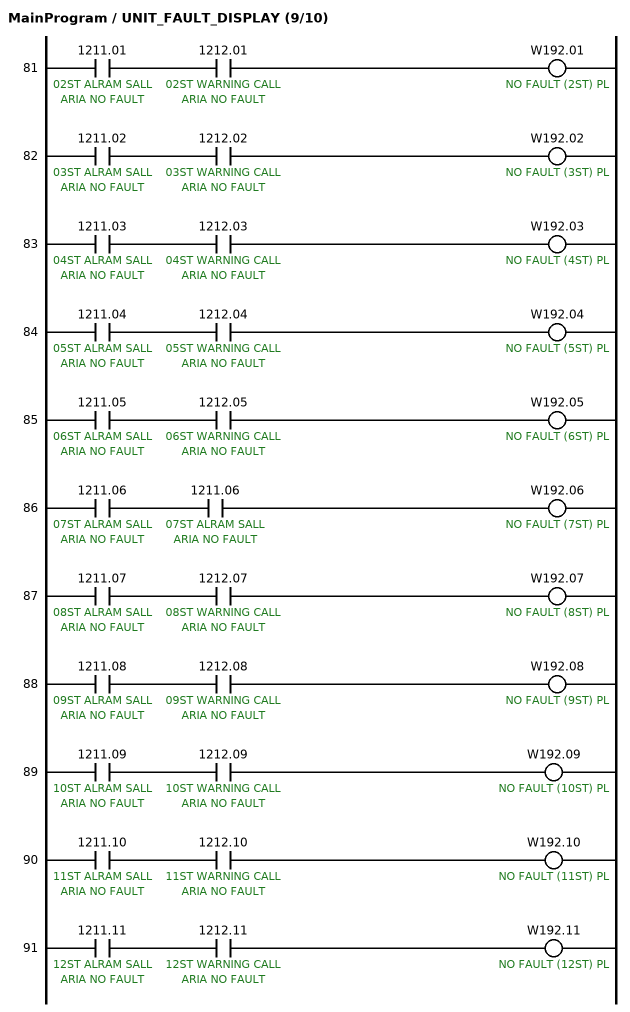
; [picture p120: MainProgram / UNIT_FAULT_DISPLAY, rungs 81-91]
; rung 81
LD 1211.01  ; 02ST ALRAM SALL ARIA NO FAULT
AND 1212.01  ; 02ST WARNING CALL ARIA NO FAULT
OUT W192.01  ; NO FAULT (2ST) PL
; rung 82
LD 1211.02  ; 03ST ALRAM SALL ARIA NO FAULT
AND 1212.02  ; 03ST WARNING CALL ARIA NO FAULT
OUT W192.02  ; NO FAULT (3ST) PL
; rung 83
LD 1211.03  ; 04ST ALRAM SALL ARIA NO FAULT
AND 1212.03  ; 04ST WARNING CALL ARIA NO FAULT
OUT W192.03  ; NO FAULT (4ST) PL
; rung 84
LD 1211.04  ; 05ST ALRAM SALL ARIA NO FAULT
AND 1212.04  ; 05ST WARNING CALL ARIA NO FAULT
OUT W192.04  ; NO FAULT (5ST) PL
; rung 85
LD 1211.05  ; 06ST ALRAM SALL ARIA NO FAULT
AND 1212.05  ; 06ST WARNING CALL ARIA NO FAULT
OUT W192.05  ; NO FAULT (6ST) PL
; rung 86
LD 1211.06  ; 07ST ALRAM SALL ARIA NO FAULT
AND 1211.06  ; 07ST ALRAM SALL ARIA NO FAULT
OUT W192.06  ; NO FAULT (7ST) PL
; rung 87
LD 1211.07  ; 08ST ALRAM SALL ARIA NO FAULT
AND 1212.07  ; 08ST WARNING CALL ARIA NO FAULT
OUT W192.07  ; NO FAULT (8ST) PL
; rung 88
LD 1211.08  ; 09ST ALRAM SALL ARIA NO FAULT
AND 1212.08  ; 09ST WARNING CALL ARIA NO FAULT
OUT W192.08  ; NO FAULT (9ST) PL
; rung 89
LD 1211.09  ; 10ST ALRAM SALL ARIA NO FAULT
AND 1212.09  ; 10ST WARNING CALL ARIA NO FAULT
OUT W192.09  ; NO FAULT (10ST) PL
; rung 90
LD 1211.10  ; 11ST ALRAM SALL ARIA NO FAULT
AND 1212.10  ; 11ST WARNING CALL ARIA NO FAULT
OUT W192.10  ; NO FAULT (11ST) PL
; rung 91
LD 1211.11  ; 12ST ALRAM SALL ARIA NO FAULT
AND 1212.11  ; 12ST WARNING CALL ARIA NO FAULT
OUT W192.11  ; NO FAULT (12ST) PL

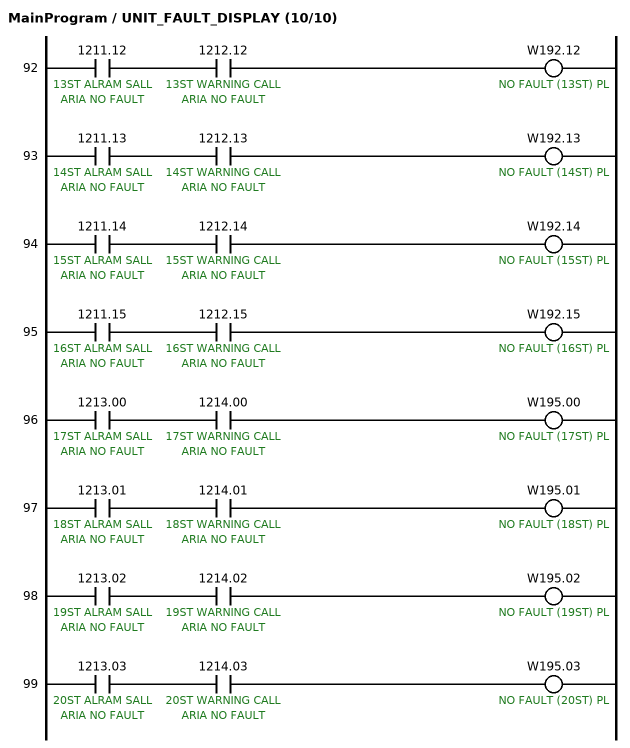
; rung 92
LD 1211.12  ; 13ST ALRAM SALL ARIA NO FAULT
AND 1212.12  ; 13ST WARNING CALL ARIA NO FAULT
OUT W192.12  ; NO FAULT (13ST) PL
; rung 93
LD 1211.13  ; 14ST ALRAM SALL ARIA NO FAULT
AND 1212.13  ; 14ST WARNING CALL ARIA NO FAULT
OUT W192.13  ; NO FAULT (14ST) PL
; rung 94
LD 1211.14  ; 15ST ALRAM SALL ARIA NO FAULT
AND 1212.14  ; 15ST WARNING CALL ARIA NO FAULT
OUT W192.14  ; NO FAULT (15ST) PL
; rung 95
LD 1211.15  ; 16ST ALRAM SALL ARIA NO FAULT
AND 1212.15  ; 16ST WARNING CALL ARIA NO FAULT
OUT W192.15  ; NO FAULT (16ST) PL
; rung 96
LD 1213.00  ; 17ST ALRAM SALL ARIA NO FAULT
AND 1214.00  ; 17ST WARNING CALL ARIA NO FAULT
OUT W195.00  ; NO FAULT (17ST) PL
; rung 97
LD 1213.01  ; 18ST ALRAM SALL ARIA NO FAULT
AND 1214.01  ; 18ST WARNING CALL ARIA NO FAULT
OUT W195.01  ; NO FAULT (18ST) PL
; rung 98
LD 1213.02  ; 19ST ALRAM SALL ARIA NO FAULT
AND 1214.02  ; 19ST WARNING CALL ARIA NO FAULT
OUT W195.02  ; NO FAULT (19ST) PL
; rung 99
LD 1213.03  ; 20ST ALRAM SALL ARIA NO FAULT
AND 1214.03  ; 20ST WARNING CALL ARIA NO FAULT
OUT W195.03  ; NO FAULT (20ST) PL

### Section FAULT_DISPLAY

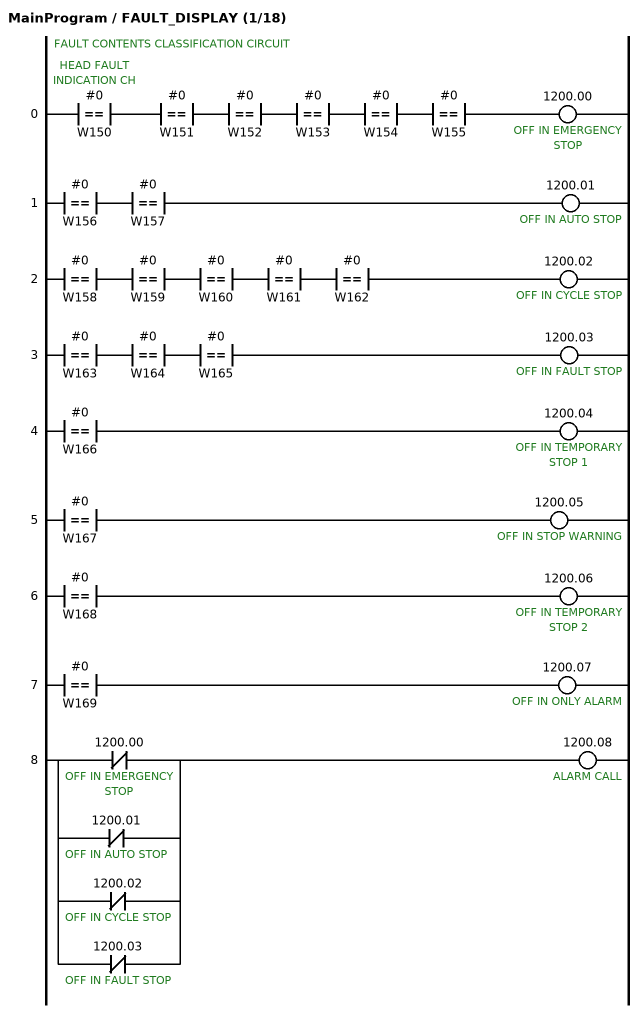
; rung 0: FAULT CONTENTS CLASSIFICATION CIRCUIT
LD=(300) #0 W150  ; HEAD FAULT INDICATION CH
AND=(300) #0 W151
AND=(300) #0 W152
AND=(300) #0 W153
AND=(300) #0 W154
AND=(300) #0 W155
OUT 1200.00  ; OFF IN EMERGENCY STOP
; rung 1
LD=(300) #0 W156
AND=(300) #0 W157
OUT 1200.01  ; OFF IN AUTO STOP
; rung 2
LD=(300) #0 W158
AND=(300) #0 W159
AND=(300) #0 W160
AND=(300) #0 W161
AND=(300) #0 W162
OUT 1200.02  ; OFF IN CYCLE STOP
; rung 3
LD=(300) #0 W163
AND=(300) #0 W164
AND=(300) #0 W165
OUT 1200.03  ; OFF IN FAULT STOP
; rung 4
LD=(300) #0 W166
OUT 1200.04  ; OFF IN TEMPORARY STOP 1
; rung 5
LD=(300) #0 W167
OUT 1200.05  ; OFF IN STOP WARNING
; rung 6
LD=(300) #0 W168
OUT 1200.06  ; OFF IN TEMPORARY STOP 2
; rung 7
LD=(300) #0 W169
OUT 1200.07  ; OFF IN ONLY ALARM
; rung 8
LDNOT 1200.00  ; OFF IN EMERGENCY STOP
ORNOT 1200.01  ; OFF IN AUTO STOP
ORNOT 1200.02  ; OFF IN CYCLE STOP
ORNOT 1200.03  ; OFF IN FAULT STOP
OUT 1200.08  ; ALARM CALL

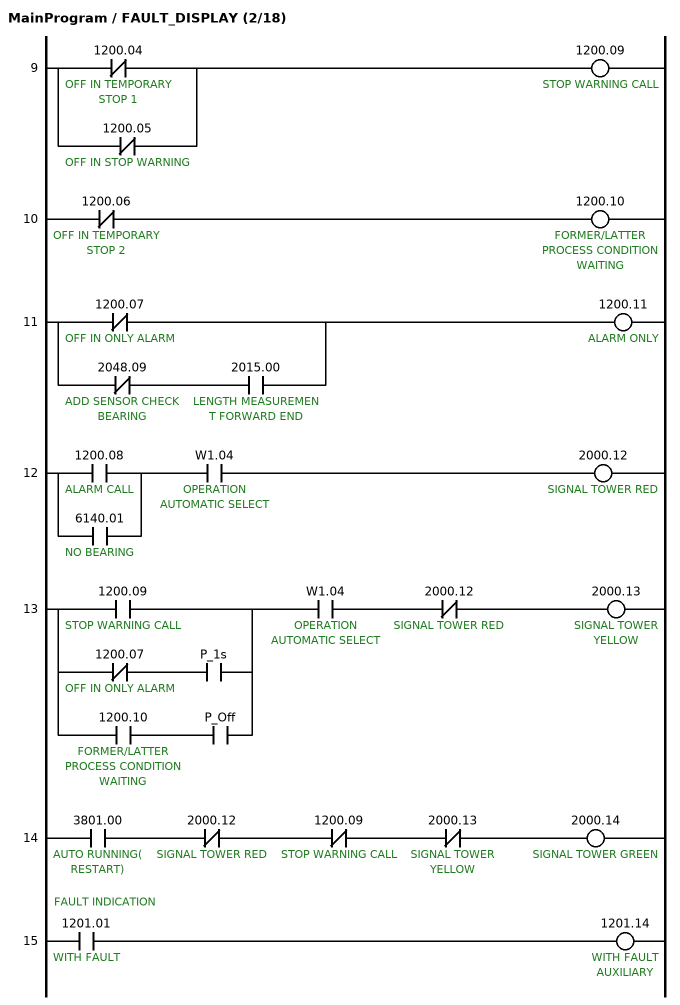
; rung 9
LDNOT 1200.04  ; OFF IN TEMPORARY STOP 1
ORNOT 1200.05  ; OFF IN STOP WARNING
OUT 1200.09  ; STOP WARNING CALL
; rung 10
LDNOT 1200.06  ; OFF IN TEMPORARY STOP 2
OUT 1200.10  ; FORMER/LATTER PROCESS CONDITION WAITING
; rung 11
LDNOT 1200.07  ; OFF IN ONLY ALARM
LDNOT 2048.09  ; ADD SENSOR CHECK BEARING
AND 2015.00  ; LENGTH MEASUREMENT FORWARD END
ORLD
OUT 1200.11  ; ALARM ONLY
; rung 12
LD 1200.08  ; ALARM CALL
OR 6140.01  ; NO BEARING
AND W1.04  ; OPERATION AUTOMATIC SELECT
OUT 2000.12  ; SIGNAL TOWER RED
; rung 13
LD 1200.09  ; STOP WARNING CALL
LDNOT 1200.07  ; OFF IN ONLY ALARM
AND P_1s
ORLD
LD 1200.10  ; FORMER/LATTER PROCESS CONDITION WAITING
AND P_Off
ORLD
AND W1.04  ; OPERATION AUTOMATIC SELECT
ANDNOT 2000.12  ; SIGNAL TOWER RED
OUT 2000.13  ; SIGNAL TOWER YELLOW
; rung 14
LD 3801.00  ; AUTO RUNNING(RESTART)
ANDNOT 2000.12  ; SIGNAL TOWER RED
ANDNOT 1200.09  ; STOP WARNING CALL
ANDNOT 2000.13  ; SIGNAL TOWER YELLOW
OUT 2000.14  ; SIGNAL TOWER GREEN
; rung 15: FAULT INDICATION
LD 1201.01  ; WITH FAULT
OUT 1201.14  ; WITH FAULT AUXILIARY

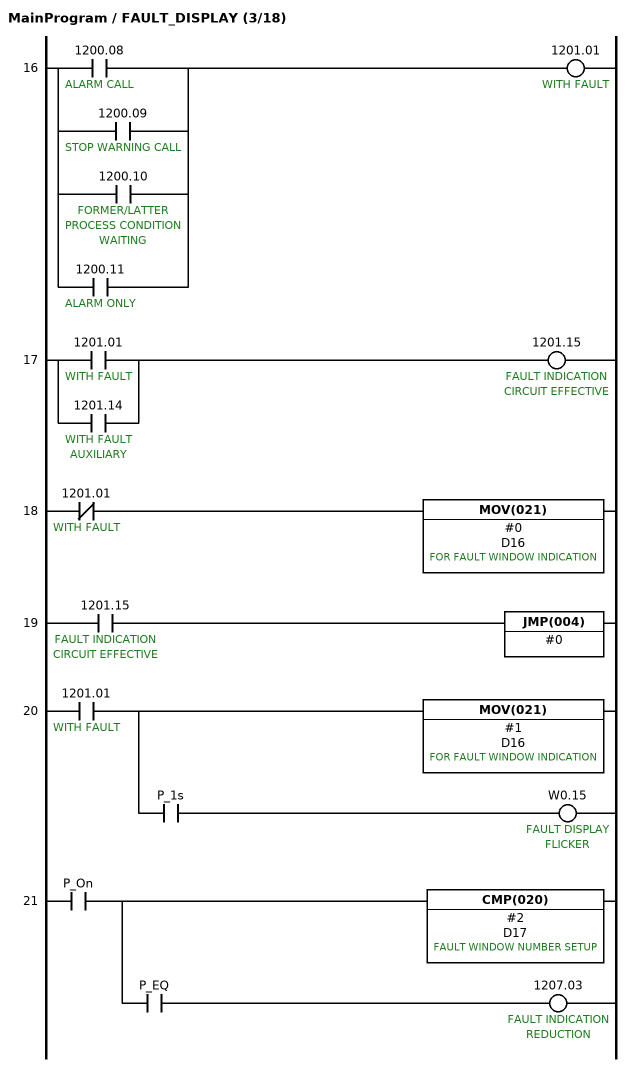
; rung 16
LD 1200.08  ; ALARM CALL
OR 1200.09  ; STOP WARNING CALL
OR 1200.10  ; FORMER/LATTER PROCESS CONDITION WAITING
OR 1200.11  ; ALARM ONLY
OUT 1201.01  ; WITH FAULT
; rung 17
LD 1201.01  ; WITH FAULT
OR 1201.14  ; WITH FAULT AUXILIARY
OUT 1201.15  ; FAULT INDICATION CIRCUIT EFFECTIVE
; rung 18
LDNOT 1201.01  ; WITH FAULT
MOV(021) #0 D16  ; FOR FAULT WINDOW INDICATION  // WITH NO FAULT WINDOW DISPLAY
; rung 19
LD 1201.15  ; FAULT INDICATION CIRCUIT EFFECTIVE
JMP(004) #0
; rung 20
LD 1201.01  ; WITH FAULT
MOV(021) #1 D16  ; FOR FAULT WINDOW INDICATION  // FAULT WINDOW DISPLAY
AND P_1s
OUT W0.15  ; FAULT DISPLAY FLICKER
; rung 21
LD P_On
CMP(020) #2 D17  ; FAULT WINDOW NUMBER SETUP
AND P_EQ
OUT 1207.03  ; FAULT INDICATION REDUCTION

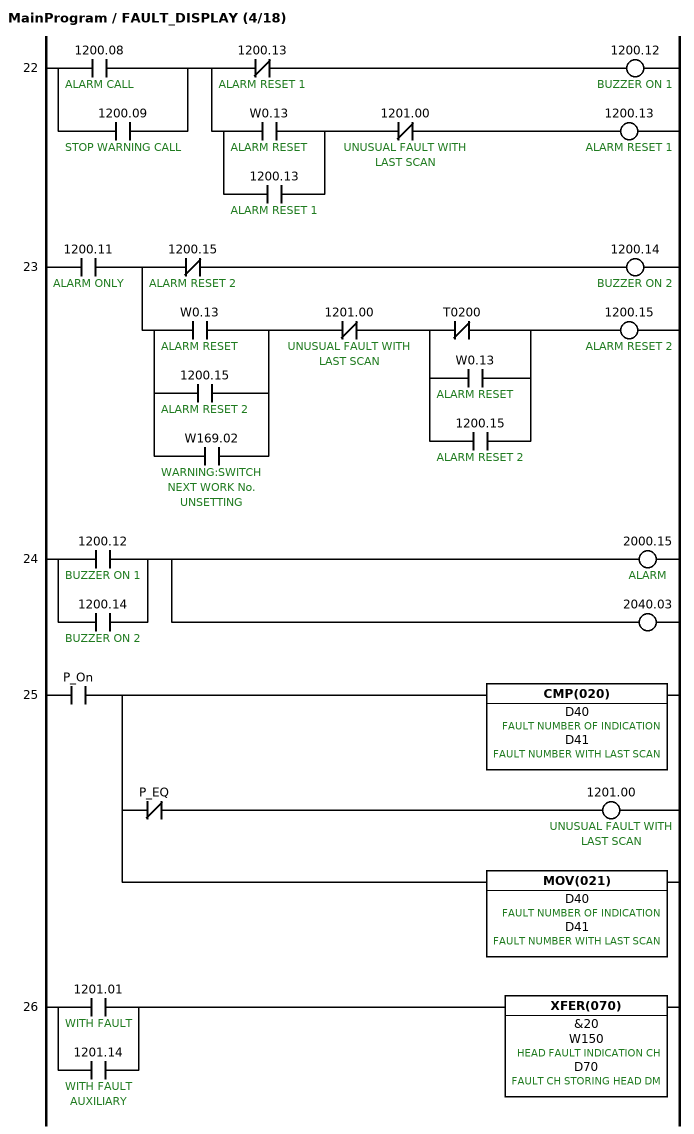
; rung 22
LD 1200.08  ; ALARM CALL
OR 1200.09  ; STOP WARNING CALL
OUT TR0
ANDNOT 1200.13  ; ALARM RESET 1
OUT 1200.12  ; BUZZER ON 1
LD TR0
LD W0.13  ; ALARM RESET
OR 1200.13  ; ALARM RESET 1
ANDLD
ANDNOT 1201.00  ; UNUSUAL FAULT WITH LAST SCAN
OUT 1200.13  ; ALARM RESET 1
; rung 23
LD 1200.11  ; ALARM ONLY
OUT TR0
ANDNOT 1200.15  ; ALARM RESET 2
OUT 1200.14  ; BUZZER ON 2
LD TR0
LD W0.13  ; ALARM RESET
OR 1200.15  ; ALARM RESET 2
OR W169.02  ; WARNING:SWITCH NEXT WORK No. UNSETTING
ANDLD
ANDNOT 1201.00  ; UNUSUAL FAULT WITH LAST SCAN
LDNOT T0200
OR W0.13  ; ALARM RESET
OR 1200.15  ; ALARM RESET 2
ANDLD
OUT 1200.15  ; ALARM RESET 2
; rung 24
LD 1200.12  ; BUZZER ON 1
OR 1200.14  ; BUZZER ON 2
OUT 2000.15  ; ALARM
OUT 2040.03
; rung 25
LD P_On
OUT TR0
CMP(020) D40 D41  ; FAULT NUMBER OF INDICATION, FAULT NUMBER WITH LAST SCAN  // FAULT NUMBER COMPARISON
ANDNOT P_EQ
OUT 1201.00  ; UNUSUAL FAULT WITH LAST SCAN
LD TR0
MOV(021) D40 D41  ; FAULT NUMBER OF INDICATION, FAULT NUMBER WITH LAST SCAN  // FAULT NUMBER TRANSMISSION FOR NEXT SCAN COMPARISON
; rung 26
LD 1201.01  ; WITH FAULT
OR 1201.14  ; WITH FAULT AUXILIARY
XFER(070) &20 W150 D70  ; HEAD FAULT INDICATION CH, FAULT CH STORING HEAD DM  // ALL FAULT CH ARE TRANSMISSION TO DM0070-89

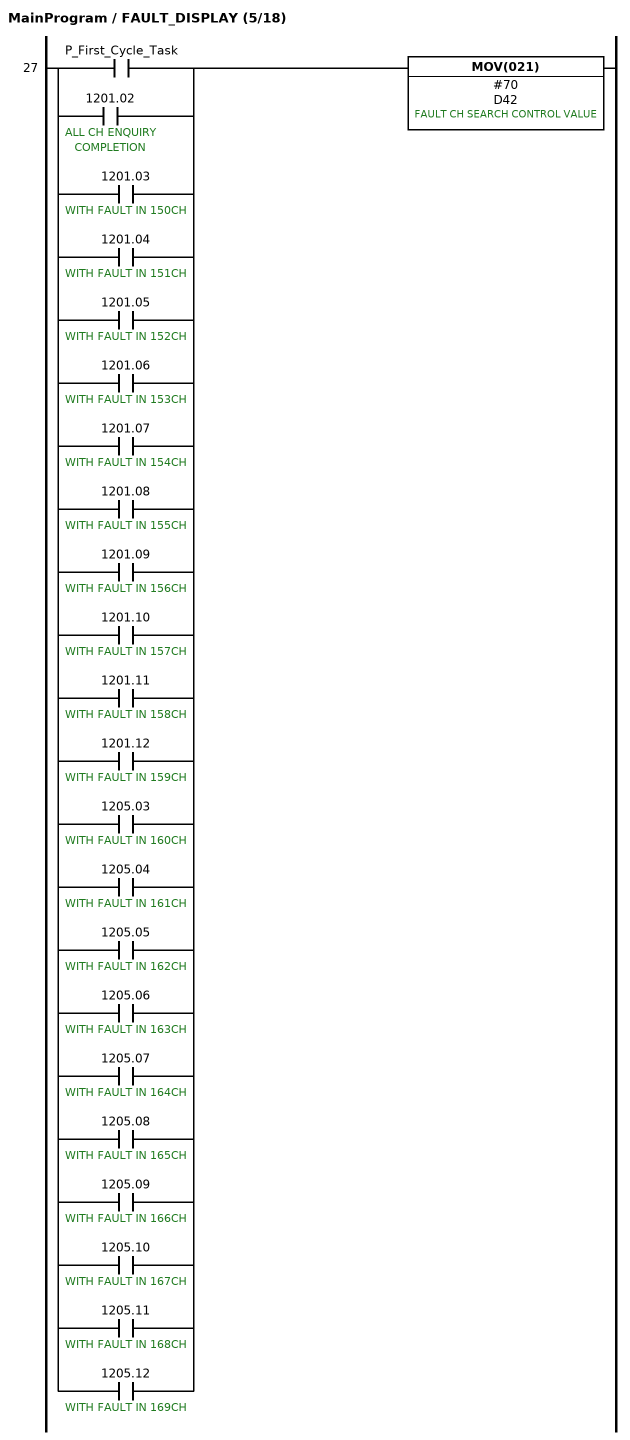
; rung 27
LD P_First_Cycle_Task
OR 1201.02  ; ALL CH ENQUIRY COMPLETION
OR 1201.03  ; WITH FAULT IN 150CH
OR 1201.04  ; WITH FAULT IN 151CH
OR 1201.05  ; WITH FAULT IN 152CH
OR 1201.06  ; WITH FAULT IN 153CH
OR 1201.07  ; WITH FAULT IN 154CH
OR 1201.08  ; WITH FAULT IN 155CH
OR 1201.09  ; WITH FAULT IN 156CH
OR 1201.10  ; WITH FAULT IN 157CH
OR 1201.11  ; WITH FAULT IN 158CH
OR 1201.12  ; WITH FAULT IN 159CH
OR 1205.03  ; WITH FAULT IN 160CH
OR 1205.04  ; WITH FAULT IN 161CH
OR 1205.05  ; WITH FAULT IN 162CH
OR 1205.06  ; WITH FAULT IN 163CH
OR 1205.07  ; WITH FAULT IN 164CH
OR 1205.08  ; WITH FAULT IN 165CH
OR 1205.09  ; WITH FAULT IN 166CH
OR 1205.10  ; WITH FAULT IN 167CH
OR 1205.11  ; WITH FAULT IN 168CH
OR 1205.12  ; WITH FAULT IN 169CH
MOV(021) #70 D42  ; FAULT CH SEARCH CONTROL VALUE  // FOR FAULT CH REFERENCE,CONTORL VALUE INITIALIZATION

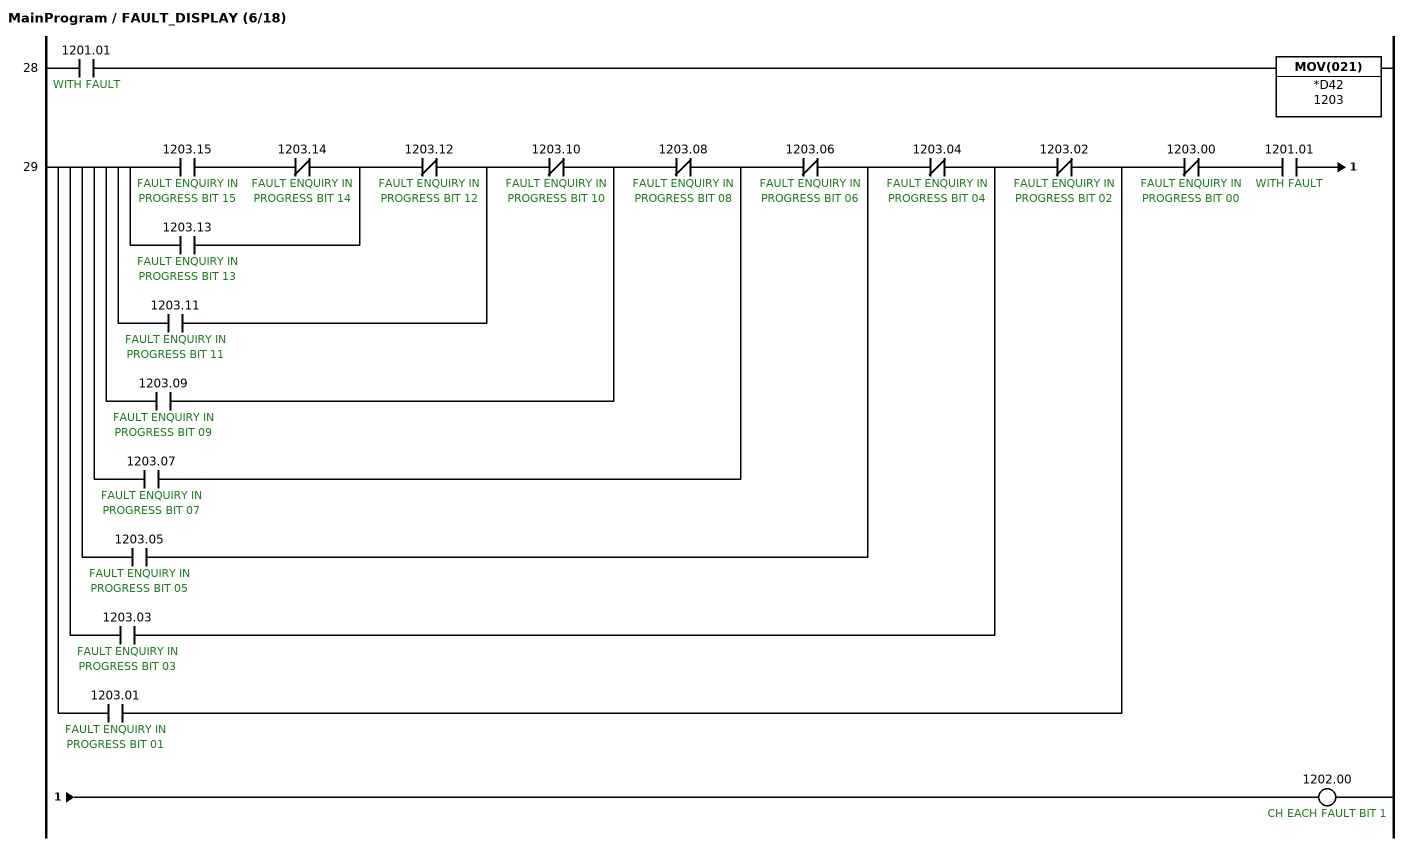
; rung 28
LD 1201.01  ; WITH FAULT
MOV(021) *D42 1203  // FAULT BIT IN CH IS TRANSMISSION DURING REFERENCE
; rung 29
LD 1203.15  ; FAULT ENQUIRY IN PROGRESS BIT 15
ANDNOT 1203.14  ; FAULT ENQUIRY IN PROGRESS BIT 14
OR 1203.13  ; FAULT ENQUIRY IN PROGRESS BIT 13
ANDNOT 1203.12  ; FAULT ENQUIRY IN PROGRESS BIT 12
OR 1203.11  ; FAULT ENQUIRY IN PROGRESS BIT 11
ANDNOT 1203.10  ; FAULT ENQUIRY IN PROGRESS BIT 10
OR 1203.09  ; FAULT ENQUIRY IN PROGRESS BIT 09
ANDNOT 1203.08  ; FAULT ENQUIRY IN PROGRESS BIT 08
OR 1203.07  ; FAULT ENQUIRY IN PROGRESS BIT 07
ANDNOT 1203.06  ; FAULT ENQUIRY IN PROGRESS BIT 06
OR 1203.05  ; FAULT ENQUIRY IN PROGRESS BIT 05
ANDNOT 1203.04  ; FAULT ENQUIRY IN PROGRESS BIT 04
OR 1203.03  ; FAULT ENQUIRY IN PROGRESS BIT 03
ANDNOT 1203.02  ; FAULT ENQUIRY IN PROGRESS BIT 02
OR 1203.01  ; FAULT ENQUIRY IN PROGRESS BIT 01
ANDNOT 1203.00  ; FAULT ENQUIRY IN PROGRESS BIT 00
AND 1201.01  ; WITH FAULT
OUT 1202.00  ; CH EACH FAULT BIT 1

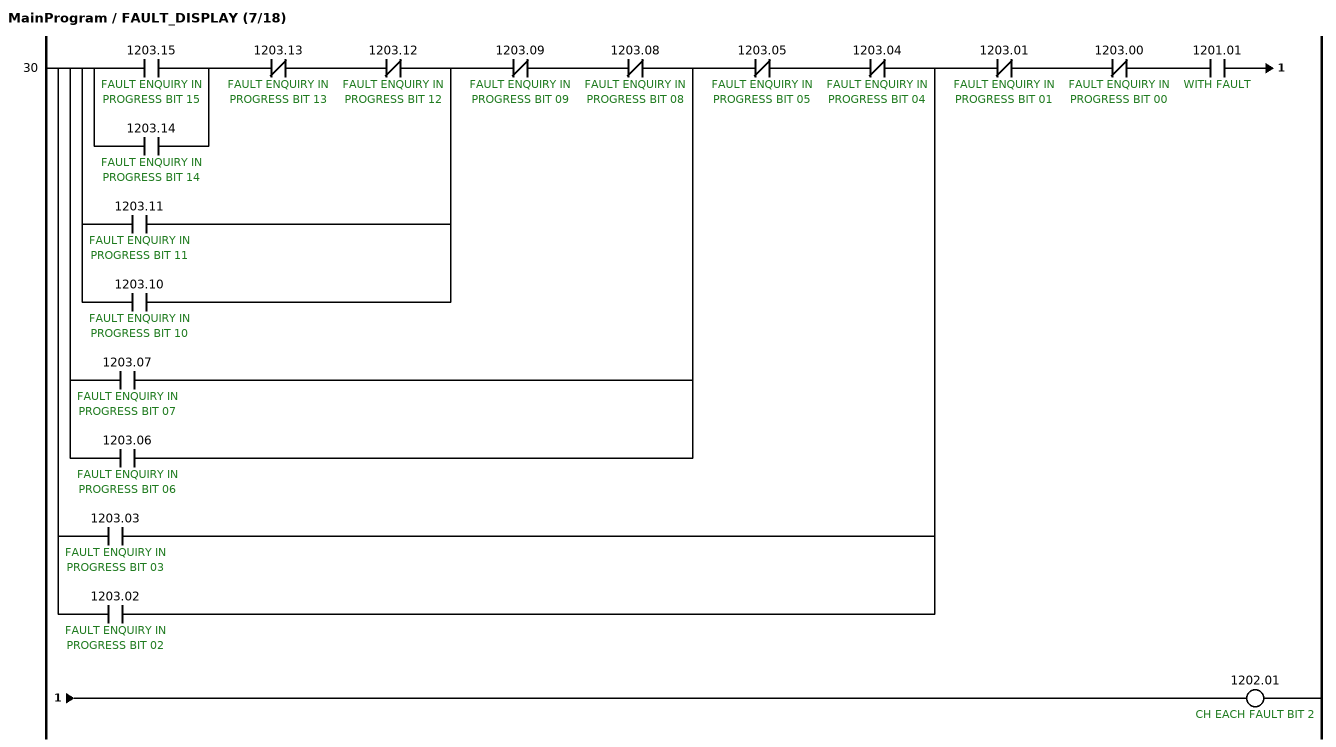
; rung 30
LD 1203.15  ; FAULT ENQUIRY IN PROGRESS BIT 15
OR 1203.14  ; FAULT ENQUIRY IN PROGRESS BIT 14
ANDNOT 1203.13  ; FAULT ENQUIRY IN PROGRESS BIT 13
ANDNOT 1203.12  ; FAULT ENQUIRY IN PROGRESS BIT 12
OR 1203.11  ; FAULT ENQUIRY IN PROGRESS BIT 11
OR 1203.10  ; FAULT ENQUIRY IN PROGRESS BIT 10
ANDNOT 1203.09  ; FAULT ENQUIRY IN PROGRESS BIT 09
ANDNOT 1203.08  ; FAULT ENQUIRY IN PROGRESS BIT 08
OR 1203.07  ; FAULT ENQUIRY IN PROGRESS BIT 07
OR 1203.06  ; FAULT ENQUIRY IN PROGRESS BIT 06
ANDNOT 1203.05  ; FAULT ENQUIRY IN PROGRESS BIT 05
ANDNOT 1203.04  ; FAULT ENQUIRY IN PROGRESS BIT 04
OR 1203.03  ; FAULT ENQUIRY IN PROGRESS BIT 03
OR 1203.02  ; FAULT ENQUIRY IN PROGRESS BIT 02
ANDNOT 1203.01  ; FAULT ENQUIRY IN PROGRESS BIT 01
ANDNOT 1203.00  ; FAULT ENQUIRY IN PROGRESS BIT 00
AND 1201.01  ; WITH FAULT
OUT 1202.01  ; CH EACH FAULT BIT 2

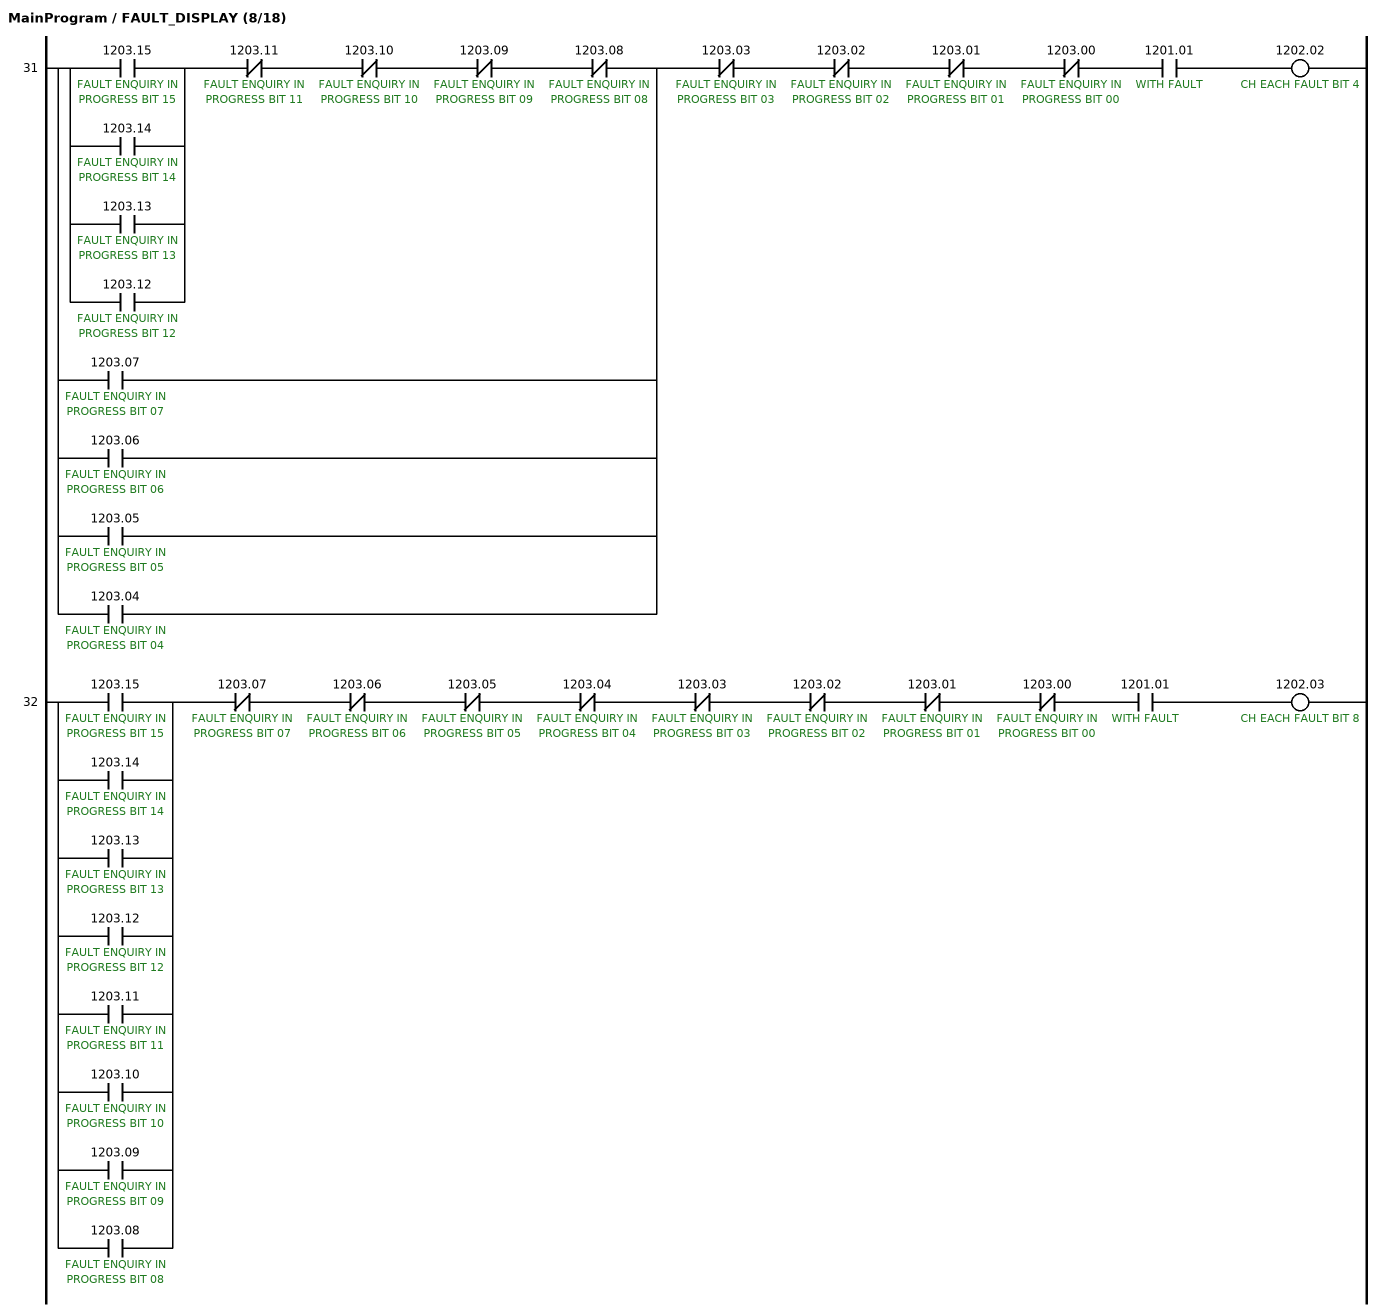
; rung 31
LD 1203.15  ; FAULT ENQUIRY IN PROGRESS BIT 15
OR 1203.14  ; FAULT ENQUIRY IN PROGRESS BIT 14
OR 1203.13  ; FAULT ENQUIRY IN PROGRESS BIT 13
OR 1203.12  ; FAULT ENQUIRY IN PROGRESS BIT 12
ANDNOT 1203.11  ; FAULT ENQUIRY IN PROGRESS BIT 11
ANDNOT 1203.10  ; FAULT ENQUIRY IN PROGRESS BIT 10
ANDNOT 1203.09  ; FAULT ENQUIRY IN PROGRESS BIT 09
ANDNOT 1203.08  ; FAULT ENQUIRY IN PROGRESS BIT 08
OR 1203.07  ; FAULT ENQUIRY IN PROGRESS BIT 07
OR 1203.06  ; FAULT ENQUIRY IN PROGRESS BIT 06
OR 1203.05  ; FAULT ENQUIRY IN PROGRESS BIT 05
OR 1203.04  ; FAULT ENQUIRY IN PROGRESS BIT 04
ANDNOT 1203.03  ; FAULT ENQUIRY IN PROGRESS BIT 03
ANDNOT 1203.02  ; FAULT ENQUIRY IN PROGRESS BIT 02
ANDNOT 1203.01  ; FAULT ENQUIRY IN PROGRESS BIT 01
ANDNOT 1203.00  ; FAULT ENQUIRY IN PROGRESS BIT 00
AND 1201.01  ; WITH FAULT
OUT 1202.02  ; CH EACH FAULT BIT 4
; rung 32
LD 1203.15  ; FAULT ENQUIRY IN PROGRESS BIT 15
OR 1203.14  ; FAULT ENQUIRY IN PROGRESS BIT 14
OR 1203.13  ; FAULT ENQUIRY IN PROGRESS BIT 13
OR 1203.12  ; FAULT ENQUIRY IN PROGRESS BIT 12
OR 1203.11  ; FAULT ENQUIRY IN PROGRESS BIT 11
OR 1203.10  ; FAULT ENQUIRY IN PROGRESS BIT 10
OR 1203.09  ; FAULT ENQUIRY IN PROGRESS BIT 09
OR 1203.08  ; FAULT ENQUIRY IN PROGRESS BIT 08
ANDNOT 1203.07  ; FAULT ENQUIRY IN PROGRESS BIT 07
ANDNOT 1203.06  ; FAULT ENQUIRY IN PROGRESS BIT 06
ANDNOT 1203.05  ; FAULT ENQUIRY IN PROGRESS BIT 05
ANDNOT 1203.04  ; FAULT ENQUIRY IN PROGRESS BIT 04
ANDNOT 1203.03  ; FAULT ENQUIRY IN PROGRESS BIT 03
ANDNOT 1203.02  ; FAULT ENQUIRY IN PROGRESS BIT 02
ANDNOT 1203.01  ; FAULT ENQUIRY IN PROGRESS BIT 01
ANDNOT 1203.00  ; FAULT ENQUIRY IN PROGRESS BIT 00
AND 1201.01  ; WITH FAULT
OUT 1202.03  ; CH EACH FAULT BIT 8

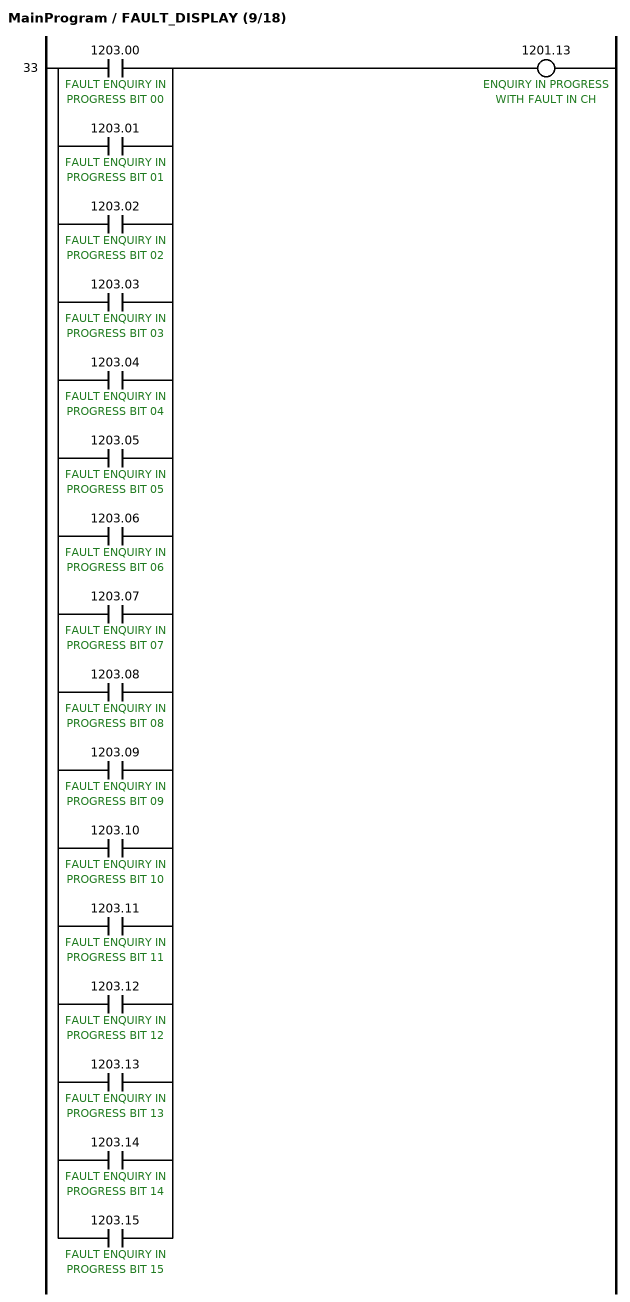
; rung 33
LD 1203.00  ; FAULT ENQUIRY IN PROGRESS BIT 00
OR 1203.01  ; FAULT ENQUIRY IN PROGRESS BIT 01
OR 1203.02  ; FAULT ENQUIRY IN PROGRESS BIT 02
OR 1203.03  ; FAULT ENQUIRY IN PROGRESS BIT 03
OR 1203.04  ; FAULT ENQUIRY IN PROGRESS BIT 04
OR 1203.05  ; FAULT ENQUIRY IN PROGRESS BIT 05
OR 1203.06  ; FAULT ENQUIRY IN PROGRESS BIT 06
OR 1203.07  ; FAULT ENQUIRY IN PROGRESS BIT 07
OR 1203.08  ; FAULT ENQUIRY IN PROGRESS BIT 08
OR 1203.09  ; FAULT ENQUIRY IN PROGRESS BIT 09
OR 1203.10  ; FAULT ENQUIRY IN PROGRESS BIT 10
OR 1203.11  ; FAULT ENQUIRY IN PROGRESS BIT 11
OR 1203.12  ; FAULT ENQUIRY IN PROGRESS BIT 12
OR 1203.13  ; FAULT ENQUIRY IN PROGRESS BIT 13
OR 1203.14  ; FAULT ENQUIRY IN PROGRESS BIT 14
OR 1203.15  ; FAULT ENQUIRY IN PROGRESS BIT 15
OUT 1201.13  ; ENQUIRY IN PROGRESS WITH FAULT IN CH

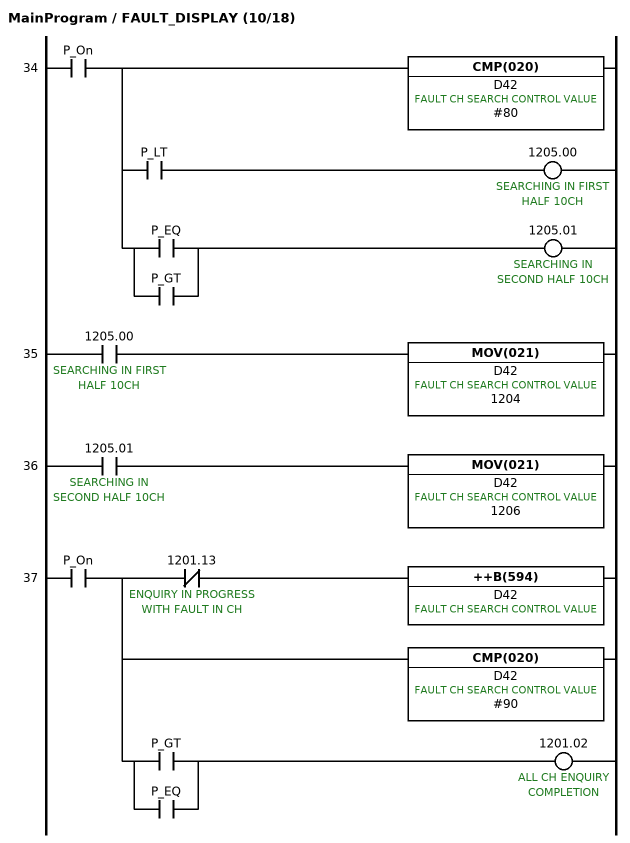
; rung 34
LD P_On
OUT TR0
CMP(020) D42 #80  ; FAULT CH SEARCH CONTROL VALUE
AND P_LT
OUT 1205.00  ; SEARCHING IN FIRST HALF 10CH
LD TR0
LD P_EQ
OR P_GT
ANDLD
OUT 1205.01  ; SEARCHING IN SECOND HALF 10CH
; rung 35
LD 1205.00  ; SEARCHING IN FIRST HALF 10CH
MOV(021) D42 1204  ; FAULT CH SEARCH CONTROL VALUE  // THE CH NUMBER WHEN BEING RETRIEVING IT IS FORWARDED.
; rung 36
LD 1205.01  ; SEARCHING IN SECOND HALF 10CH
MOV(021) D42 1206  ; FAULT CH SEARCH CONTROL VALUE  // THE CH NUMBER WHEN BEING RETRIEVING IT IS FORWARDED.
; rung 37
LD P_On
OUT TR0
ANDNOT 1201.13  ; ENQUIRY IN PROGRESS WITH FAULT IN CH
++B(594) D42  ; FAULT CH SEARCH CONTROL VALUE  // FOR REFERENCE FAULT CH,CONTROL VALUE +1
LD TR0
CMP(020) D42 #90  ; FAULT CH SEARCH CONTROL VALUE  // 90 OR MORE CONTROL VALUES FOR REFERENCE FAULT CH
LD P_GT
OR P_EQ
ANDLD
OUT 1201.02  ; ALL CH ENQUIRY COMPLETION

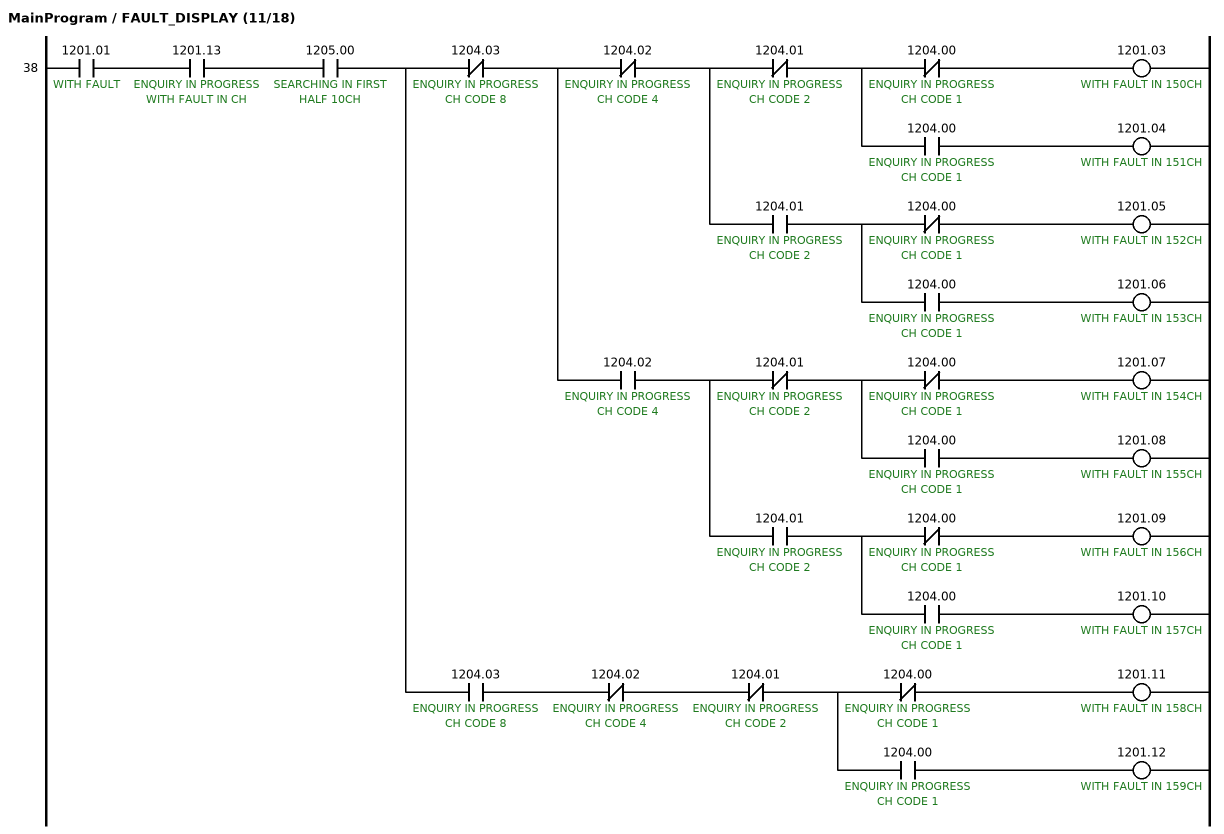
; rung 38
LD 1201.01  ; WITH FAULT
AND 1201.13  ; ENQUIRY IN PROGRESS WITH FAULT IN CH
AND 1205.00  ; SEARCHING IN FIRST HALF 10CH
OUT TR0
ANDNOT 1204.03  ; ENQUIRY IN PROGRESS CH CODE 8
OUT TR1
ANDNOT 1204.02  ; ENQUIRY IN PROGRESS CH CODE 4
OUT TR2
ANDNOT 1204.01  ; ENQUIRY IN PROGRESS CH CODE 2
OUT TR3
ANDNOT 1204.00  ; ENQUIRY IN PROGRESS CH CODE 1
OUT 1201.03  ; WITH FAULT IN 150CH
LD TR3
AND 1204.00  ; ENQUIRY IN PROGRESS CH CODE 1
OUT 1201.04  ; WITH FAULT IN 151CH
LD TR2
AND 1204.01  ; ENQUIRY IN PROGRESS CH CODE 2
OUT TR2
ANDNOT 1204.00  ; ENQUIRY IN PROGRESS CH CODE 1
OUT 1201.05  ; WITH FAULT IN 152CH
LD TR2
AND 1204.00  ; ENQUIRY IN PROGRESS CH CODE 1
OUT 1201.06  ; WITH FAULT IN 153CH
LD TR1
AND 1204.02  ; ENQUIRY IN PROGRESS CH CODE 4
OUT TR1
ANDNOT 1204.01  ; ENQUIRY IN PROGRESS CH CODE 2
OUT TR2
ANDNOT 1204.00  ; ENQUIRY IN PROGRESS CH CODE 1
OUT 1201.07  ; WITH FAULT IN 154CH
LD TR2
AND 1204.00  ; ENQUIRY IN PROGRESS CH CODE 1
OUT 1201.08  ; WITH FAULT IN 155CH
LD TR1
AND 1204.01  ; ENQUIRY IN PROGRESS CH CODE 2
OUT TR1
ANDNOT 1204.00  ; ENQUIRY IN PROGRESS CH CODE 1
OUT 1201.09  ; WITH FAULT IN 156CH
LD TR1
AND 1204.00  ; ENQUIRY IN PROGRESS CH CODE 1
OUT 1201.10  ; WITH FAULT IN 157CH
LD TR0
AND 1204.03  ; ENQUIRY IN PROGRESS CH CODE 8
ANDNOT 1204.02  ; ENQUIRY IN PROGRESS CH CODE 4
ANDNOT 1204.01  ; ENQUIRY IN PROGRESS CH CODE 2
OUT TR0
ANDNOT 1204.00  ; ENQUIRY IN PROGRESS CH CODE 1
OUT 1201.11  ; WITH FAULT IN 158CH
LD TR0
AND 1204.00  ; ENQUIRY IN PROGRESS CH CODE 1
OUT 1201.12  ; WITH FAULT IN 159CH

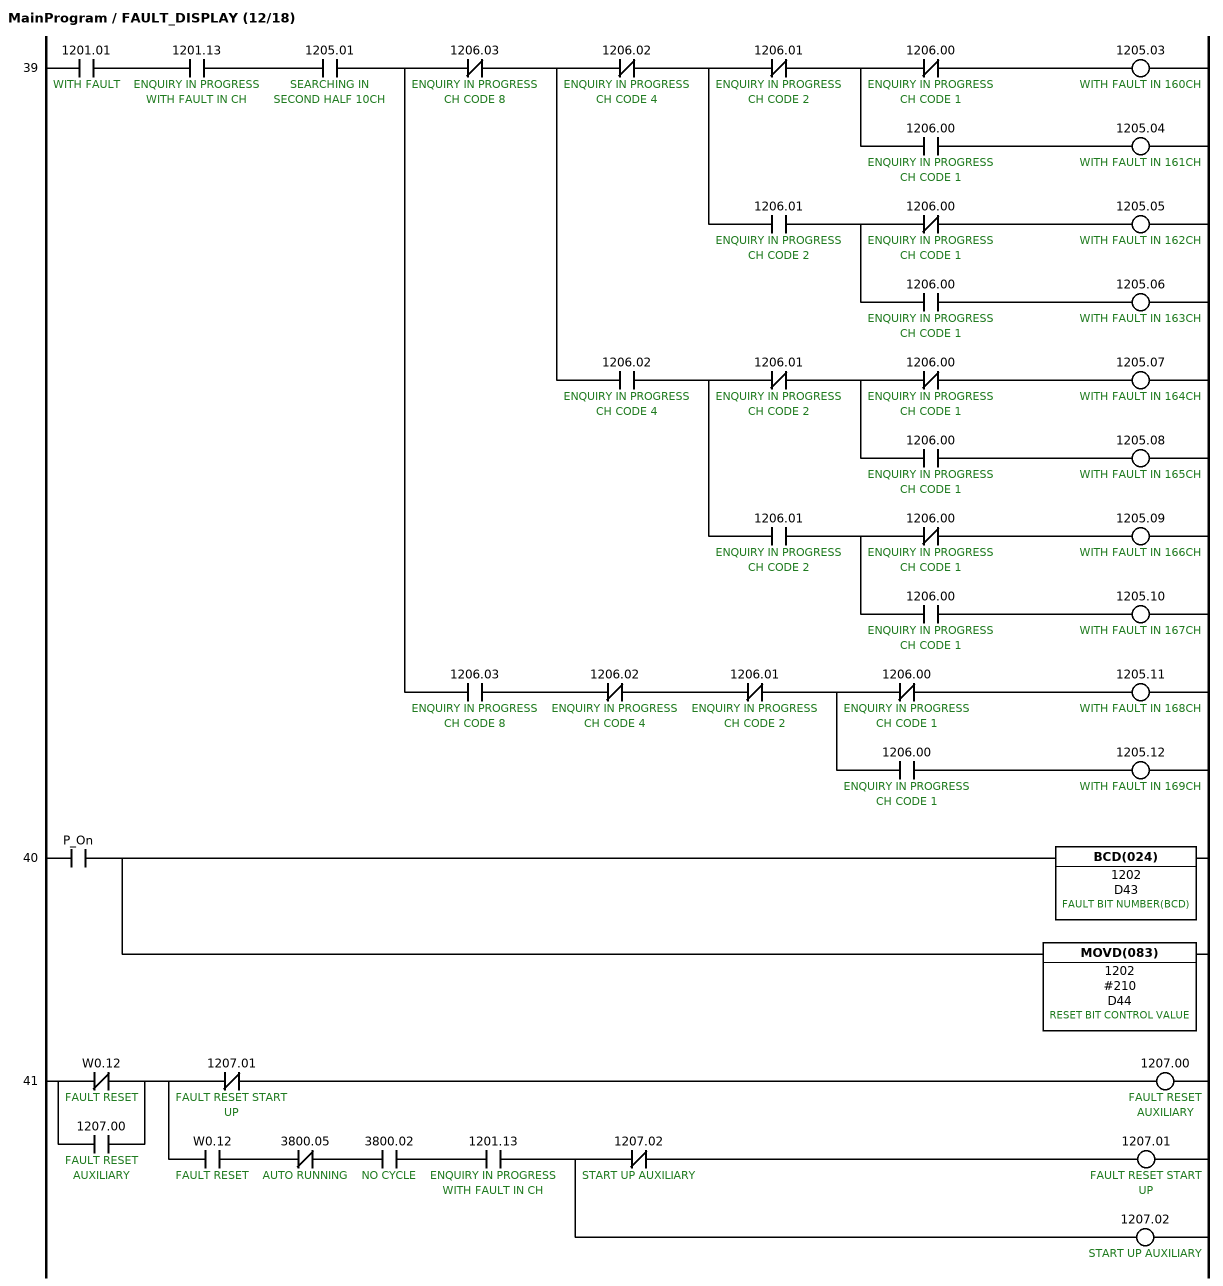
; rung 39
LD 1201.01  ; WITH FAULT
AND 1201.13  ; ENQUIRY IN PROGRESS WITH FAULT IN CH
AND 1205.01  ; SEARCHING IN SECOND HALF 10CH
OUT TR0
ANDNOT 1206.03  ; ENQUIRY IN PROGRESS CH CODE 8
OUT TR1
ANDNOT 1206.02  ; ENQUIRY IN PROGRESS CH CODE 4
OUT TR2
ANDNOT 1206.01  ; ENQUIRY IN PROGRESS CH CODE 2
OUT TR3
ANDNOT 1206.00  ; ENQUIRY IN PROGRESS CH CODE 1
OUT 1205.03  ; WITH FAULT IN 160CH
LD TR3
AND 1206.00  ; ENQUIRY IN PROGRESS CH CODE 1
OUT 1205.04  ; WITH FAULT IN 161CH
LD TR2
AND 1206.01  ; ENQUIRY IN PROGRESS CH CODE 2
OUT TR2
ANDNOT 1206.00  ; ENQUIRY IN PROGRESS CH CODE 1
OUT 1205.05  ; WITH FAULT IN 162CH
LD TR2
AND 1206.00  ; ENQUIRY IN PROGRESS CH CODE 1
OUT 1205.06  ; WITH FAULT IN 163CH
LD TR1
AND 1206.02  ; ENQUIRY IN PROGRESS CH CODE 4
OUT TR1
ANDNOT 1206.01  ; ENQUIRY IN PROGRESS CH CODE 2
OUT TR2
ANDNOT 1206.00  ; ENQUIRY IN PROGRESS CH CODE 1
OUT 1205.07  ; WITH FAULT IN 164CH
LD TR2
AND 1206.00  ; ENQUIRY IN PROGRESS CH CODE 1
OUT 1205.08  ; WITH FAULT IN 165CH
LD TR1
AND 1206.01  ; ENQUIRY IN PROGRESS CH CODE 2
OUT TR1
ANDNOT 1206.00  ; ENQUIRY IN PROGRESS CH CODE 1
OUT 1205.09  ; WITH FAULT IN 166CH
LD TR1
AND 1206.00  ; ENQUIRY IN PROGRESS CH CODE 1
OUT 1205.10  ; WITH FAULT IN 167CH
LD TR0
AND 1206.03  ; ENQUIRY IN PROGRESS CH CODE 8
ANDNOT 1206.02  ; ENQUIRY IN PROGRESS CH CODE 4
ANDNOT 1206.01  ; ENQUIRY IN PROGRESS CH CODE 2
OUT TR0
ANDNOT 1206.00  ; ENQUIRY IN PROGRESS CH CODE 1
OUT 1205.11  ; WITH FAULT IN 168CH
LD TR0
AND 1206.00  ; ENQUIRY IN PROGRESS CH CODE 1
OUT 1205.12  ; WITH FAULT IN 169CH
; rung 40
LD P_On
BCD(024) 1202 D43  ; FAULT BIT NUMBER(BCD)  // FAULT BIT No. CHANGE BCD
MOVD(083) 1202 #210 D44  ; RESET BIT CONTROL VALUE  // RESET BIT CONTROL
; rung 41
LDNOT W0.12  ; FAULT RESET
OR 1207.00  ; FAULT RESET AUXILIARY
OUT TR0
ANDNOT 1207.01  ; FAULT RESET START UP
OUT 1207.00  ; FAULT RESET AUXILIARY
LD TR0
AND W0.12  ; FAULT RESET
ANDNOT 3800.05  ; AUTO RUNNING
AND 3800.02  ; NO CYCLE
AND 1201.13  ; ENQUIRY IN PROGRESS WITH FAULT IN CH
OUT TR0
ANDNOT 1207.02  ; START UP AUXILIARY
OUT 1207.01  ; FAULT RESET START UP
LD TR0
OUT 1207.02  ; START UP AUXILIARY

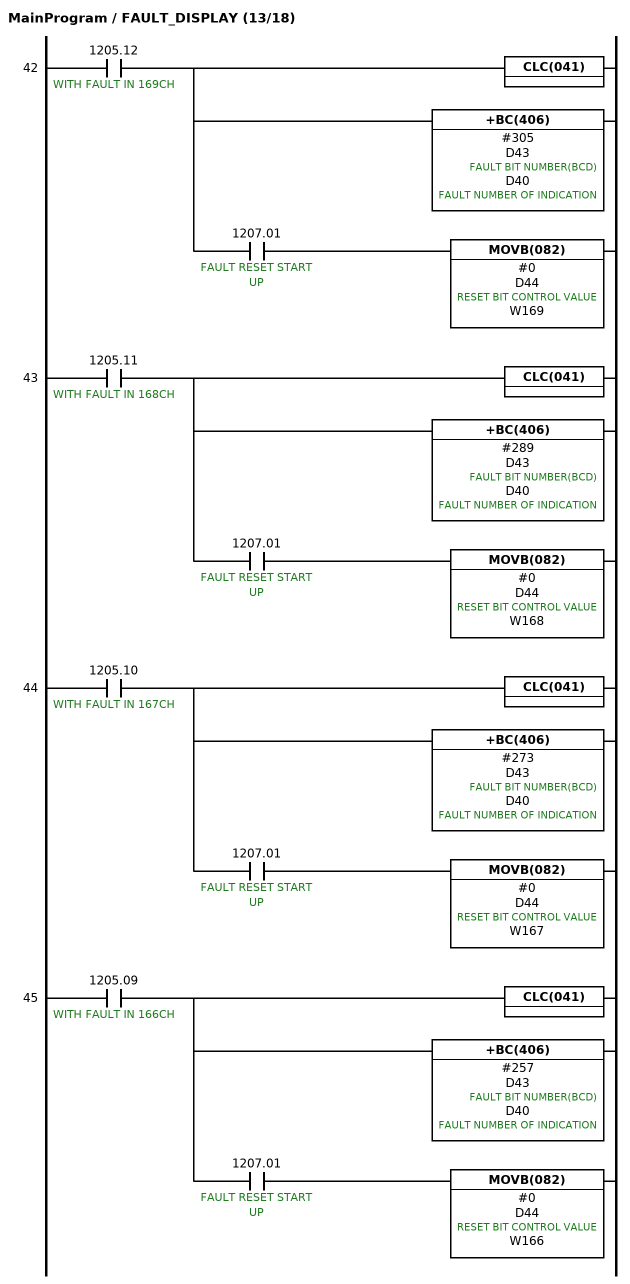
; rung 42
LD 1205.12  ; WITH FAULT IN 169CH
CLC(041)
+BC(406) #305 D43 D40  ; FAULT BIT NUMBER(BCD), FAULT NUMBER OF INDICATION  // FAULT NUMBER TRANSMISSION IN CH
AND 1207.01  ; FAULT RESET START UP
MOVB(082) #0 D44 W169  ; RESET BIT CONTROL VALUE  // FAULT BIT RESET IN CH
; rung 43
LD 1205.11  ; WITH FAULT IN 168CH
CLC(041)
+BC(406) #289 D43 D40  ; FAULT BIT NUMBER(BCD), FAULT NUMBER OF INDICATION  // FAULT NUMBER TRANSMISSION IN CH
AND 1207.01  ; FAULT RESET START UP
MOVB(082) #0 D44 W168  ; RESET BIT CONTROL VALUE  // FAULT BIT RESET IN CH
; rung 44
LD 1205.10  ; WITH FAULT IN 167CH
CLC(041)
+BC(406) #273 D43 D40  ; FAULT BIT NUMBER(BCD), FAULT NUMBER OF INDICATION  // FAULT NUMBER TRANSMISSION IN CH
AND 1207.01  ; FAULT RESET START UP
MOVB(082) #0 D44 W167  ; RESET BIT CONTROL VALUE  // FAULT BIT RESET IN CH
; rung 45
LD 1205.09  ; WITH FAULT IN 166CH
CLC(041)
+BC(406) #257 D43 D40  ; FAULT BIT NUMBER(BCD), FAULT NUMBER OF INDICATION  // FAULT NUMBER TRANSMISSION IN CH
AND 1207.01  ; FAULT RESET START UP
MOVB(082) #0 D44 W166  ; RESET BIT CONTROL VALUE  // FAULT BIT RESET IN CH

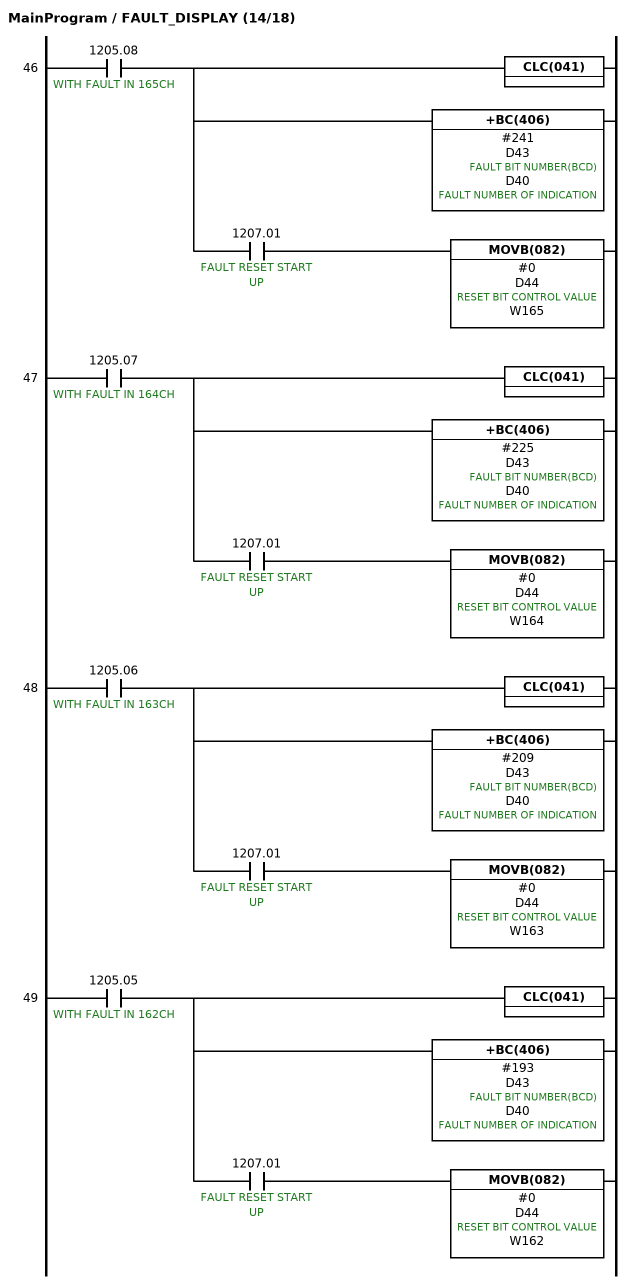
; rung 46
LD 1205.08  ; WITH FAULT IN 165CH
CLC(041)
+BC(406) #241 D43 D40  ; FAULT BIT NUMBER(BCD), FAULT NUMBER OF INDICATION  // FAULT NUMBER TRANSMISSION IN CH
AND 1207.01  ; FAULT RESET START UP
MOVB(082) #0 D44 W165  ; RESET BIT CONTROL VALUE  // FAULT BIT RESET IN CH
; rung 47
LD 1205.07  ; WITH FAULT IN 164CH
CLC(041)
+BC(406) #225 D43 D40  ; FAULT BIT NUMBER(BCD), FAULT NUMBER OF INDICATION  // FAULT NUMBER TRANSMISSION IN CH
AND 1207.01  ; FAULT RESET START UP
MOVB(082) #0 D44 W164  ; RESET BIT CONTROL VALUE  // FAULT BIT RESET IN CH
; rung 48
LD 1205.06  ; WITH FAULT IN 163CH
CLC(041)
+BC(406) #209 D43 D40  ; FAULT BIT NUMBER(BCD), FAULT NUMBER OF INDICATION  // FAULT NUMBER TRANSMISSION IN CH
AND 1207.01  ; FAULT RESET START UP
MOVB(082) #0 D44 W163  ; RESET BIT CONTROL VALUE  // FAULT BIT RESET IN CH
; rung 49
LD 1205.05  ; WITH FAULT IN 162CH
CLC(041)
+BC(406) #193 D43 D40  ; FAULT BIT NUMBER(BCD), FAULT NUMBER OF INDICATION  // FAULT NUMBER TRANSMISSION IN CH
AND 1207.01  ; FAULT RESET START UP
MOVB(082) #0 D44 W162  ; RESET BIT CONTROL VALUE  // FAULT BIT RESET IN CH

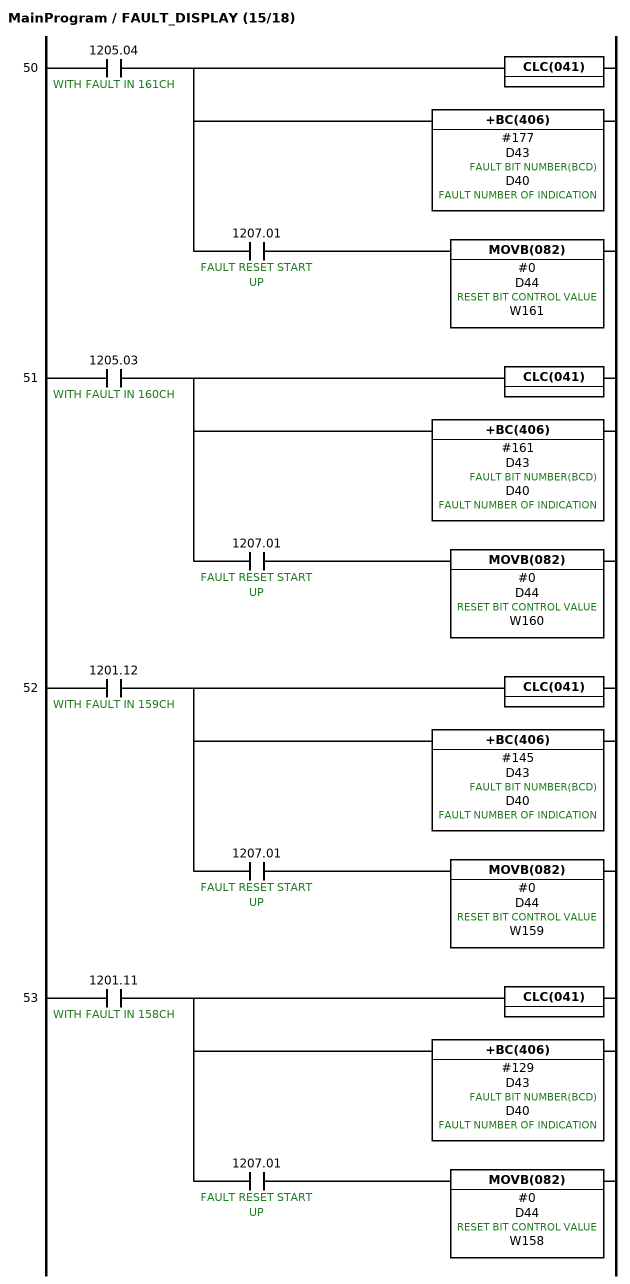
; rung 50
LD 1205.04  ; WITH FAULT IN 161CH
CLC(041)
+BC(406) #177 D43 D40  ; FAULT BIT NUMBER(BCD), FAULT NUMBER OF INDICATION  // FAULT NUMBER TRANSMISSION IN CH
AND 1207.01  ; FAULT RESET START UP
MOVB(082) #0 D44 W161  ; RESET BIT CONTROL VALUE  // FAULT BIT RESET IN CH
; rung 51
LD 1205.03  ; WITH FAULT IN 160CH
CLC(041)
+BC(406) #161 D43 D40  ; FAULT BIT NUMBER(BCD), FAULT NUMBER OF INDICATION  // FAULT NUMBER TRANSMISSION IN CH
AND 1207.01  ; FAULT RESET START UP
MOVB(082) #0 D44 W160  ; RESET BIT CONTROL VALUE  // FAULT BIT RESET IN CH
; rung 52
LD 1201.12  ; WITH FAULT IN 159CH
CLC(041)
+BC(406) #145 D43 D40  ; FAULT BIT NUMBER(BCD), FAULT NUMBER OF INDICATION  // FAULT NUMBER TRANSMISSION IN CH
AND 1207.01  ; FAULT RESET START UP
MOVB(082) #0 D44 W159  ; RESET BIT CONTROL VALUE  // FAULT BIT RESET IN CH
; rung 53
LD 1201.11  ; WITH FAULT IN 158CH
CLC(041)
+BC(406) #129 D43 D40  ; FAULT BIT NUMBER(BCD), FAULT NUMBER OF INDICATION  // FAULT NUMBER TRANSMISSION IN CH
AND 1207.01  ; FAULT RESET START UP
MOVB(082) #0 D44 W158  ; RESET BIT CONTROL VALUE  // FAULT BIT RESET IN CH

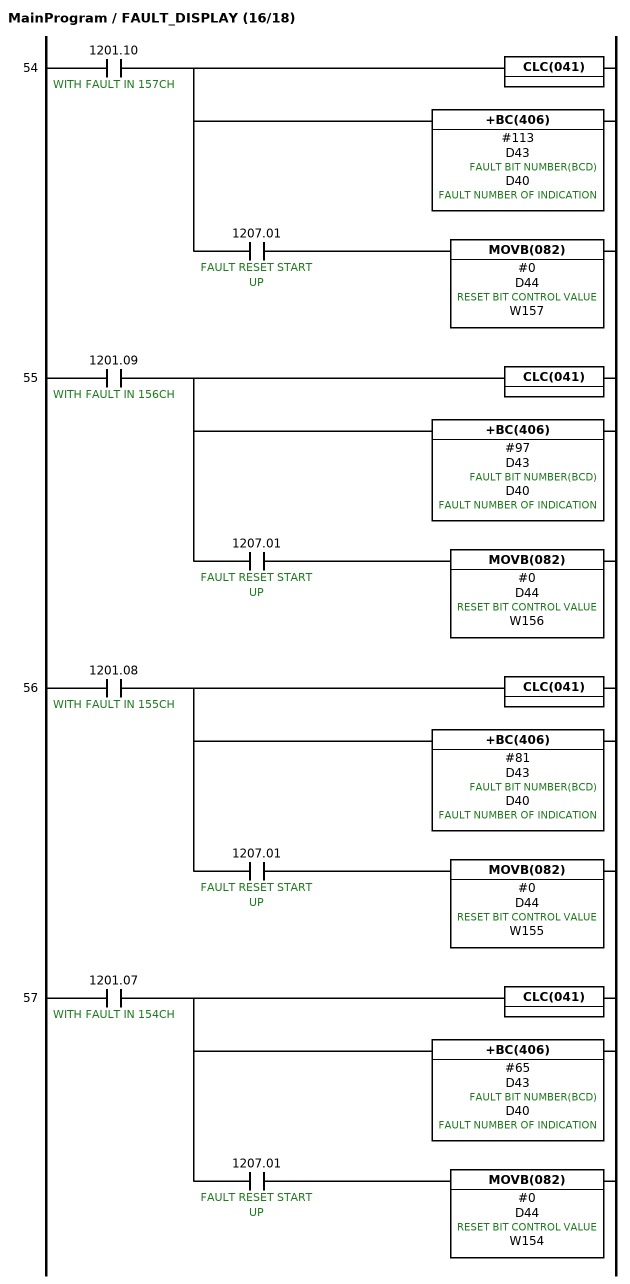
; rung 54
LD 1201.10  ; WITH FAULT IN 157CH
CLC(041)
+BC(406) #113 D43 D40  ; FAULT BIT NUMBER(BCD), FAULT NUMBER OF INDICATION  // FAULT NUMBER TRANSMISSION IN CH
AND 1207.01  ; FAULT RESET START UP
MOVB(082) #0 D44 W157  ; RESET BIT CONTROL VALUE  // FAULT BIT RESET IN CH
; rung 55
LD 1201.09  ; WITH FAULT IN 156CH
CLC(041)
+BC(406) #97 D43 D40  ; FAULT BIT NUMBER(BCD), FAULT NUMBER OF INDICATION  // FAULT NUMBER TRANSMISSION IN CH
AND 1207.01  ; FAULT RESET START UP
MOVB(082) #0 D44 W156  ; RESET BIT CONTROL VALUE  // FAULT BIT RESET IN CH
; rung 56
LD 1201.08  ; WITH FAULT IN 155CH
CLC(041)
+BC(406) #81 D43 D40  ; FAULT BIT NUMBER(BCD), FAULT NUMBER OF INDICATION  // FAULT NUMBER TRANSMISSION IN CH
AND 1207.01  ; FAULT RESET START UP
MOVB(082) #0 D44 W155  ; RESET BIT CONTROL VALUE  // FAULT BIT RESET IN CH
; rung 57
LD 1201.07  ; WITH FAULT IN 154CH
CLC(041)
+BC(406) #65 D43 D40  ; FAULT BIT NUMBER(BCD), FAULT NUMBER OF INDICATION  // FAULT NUMBER TRANSMISSION IN CH
AND 1207.01  ; FAULT RESET START UP
MOVB(082) #0 D44 W154  ; RESET BIT CONTROL VALUE  // FAULT BIT RESET IN CH

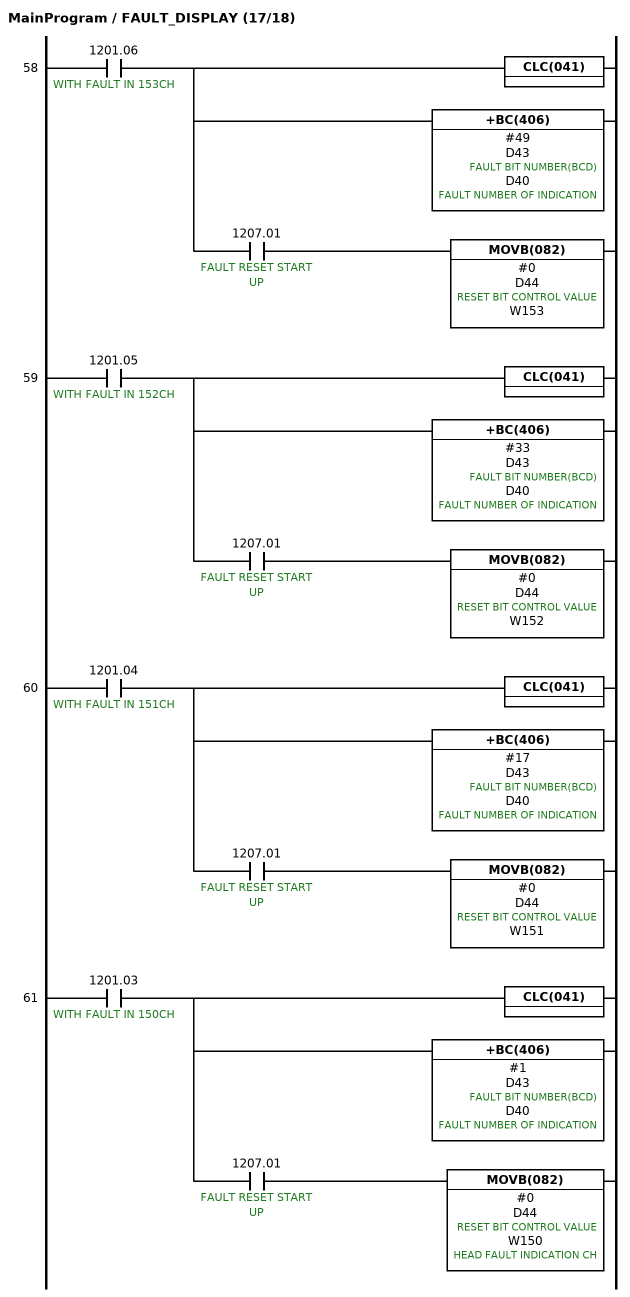
; rung 58
LD 1201.06  ; WITH FAULT IN 153CH
CLC(041)
+BC(406) #49 D43 D40  ; FAULT BIT NUMBER(BCD), FAULT NUMBER OF INDICATION  // FAULT NUMBER TRANSMISSION IN CH
AND 1207.01  ; FAULT RESET START UP
MOVB(082) #0 D44 W153  ; RESET BIT CONTROL VALUE  // FAULT BIT RESET IN CH
; rung 59
LD 1201.05  ; WITH FAULT IN 152CH
CLC(041)
+BC(406) #33 D43 D40  ; FAULT BIT NUMBER(BCD), FAULT NUMBER OF INDICATION  // FAULT NUMBER TRANSMISSION IN CH
AND 1207.01  ; FAULT RESET START UP
MOVB(082) #0 D44 W152  ; RESET BIT CONTROL VALUE  // FAULT BIT RESET IN CH
; rung 60
LD 1201.04  ; WITH FAULT IN 151CH
CLC(041)
+BC(406) #17 D43 D40  ; FAULT BIT NUMBER(BCD), FAULT NUMBER OF INDICATION  // FAULT NUMBER TRANSMISSION IN CH
AND 1207.01  ; FAULT RESET START UP
MOVB(082) #0 D44 W151  ; RESET BIT CONTROL VALUE  // FAULT BIT RESET IN CH
; rung 61
LD 1201.03  ; WITH FAULT IN 150CH
CLC(041)
+BC(406) #1 D43 D40  ; FAULT BIT NUMBER(BCD), FAULT NUMBER OF INDICATION  // FAULT NUMBER TRANSMISSION IN CH
AND 1207.01  ; FAULT RESET START UP
MOVB(082) #0 D44 W150  ; RESET BIT CONTROL VALUE, HEAD FAULT INDICATION CH  // FAULT BIT RESET IN CH

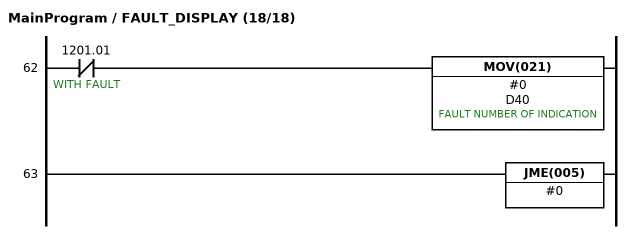
; rung 62
LDNOT 1201.01  ; WITH FAULT
MOV(021) #0 D40  ; FAULT NUMBER OF INDICATION  // FAULT NUMBER CLEARANCE WITHOUT NO FAULT
; rung 63
JME(005) #0

### Section COUNT

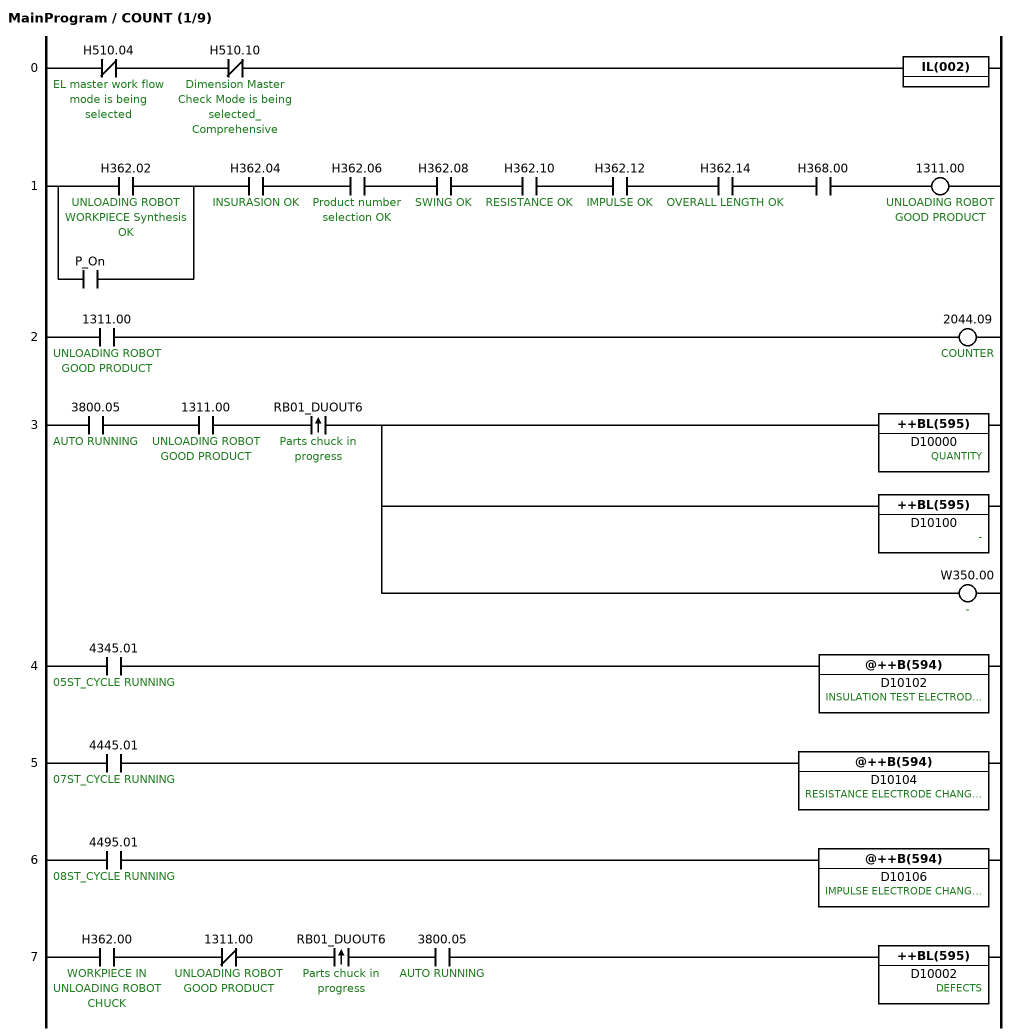
; rung 0
LDNOT H510.04  ; EL master work flow mode is being selected
ANDNOT H510.10  ; Dimension Master Check Mode is being selected_Comprehensive
IL(002)
; rung 1
LD H362.02  ; UNLOADING ROBOT WORKPIECE Synthesis OK
OR P_On
AND H362.04  ; INSURASION OK
AND H362.06  ; Product number selection OK
AND H362.08  ; SWING OK
AND H362.10  ; RESISTANCE OK
AND H362.12  ; IMPULSE OK
AND H362.14  ; OVERALL LENGTH OK
AND H368.00
OUT 1311.00  ; UNLOADING ROBOT GOOD PRODUCT
; rung 2
LD 1311.00  ; UNLOADING ROBOT GOOD PRODUCT
OUT 2044.09  ; COUNTER
; rung 3
LD 3800.05  ; AUTO RUNNING
AND 1311.00  ; UNLOADING ROBOT GOOD PRODUCT
@AND RB01_DUOUT6  ; Parts chuck in progress
++BL(595) D10000  ; QUANTITY
++BL(595) D10100  ; -
OUT W350.00  ; -
; rung 4
LD 4345.01  ; 05ST_CYCLE RUNNING
@++B(594) D10102  ; INSULATION TEST ELECTRODE CHANGE PRESENT
; rung 5
LD 4445.01  ; 07ST_CYCLE RUNNING
@++B(594) D10104  ; RESISTANCE ELECTRODE CHANGE PRESENT
; rung 6
LD 4495.01  ; 08ST_CYCLE RUNNING
@++B(594) D10106  ; IMPULSE ELECTRODE CHANGE PRESENT
; rung 7
LD H362.00  ; WORKPIECE IN UNLOADING ROBOT CHUCK
ANDNOT 1311.00  ; UNLOADING ROBOT GOOD PRODUCT
@AND RB01_DUOUT6  ; Parts chuck in progress
AND 3800.05  ; AUTO RUNNING
++BL(595) D10002  ; DEFECTS

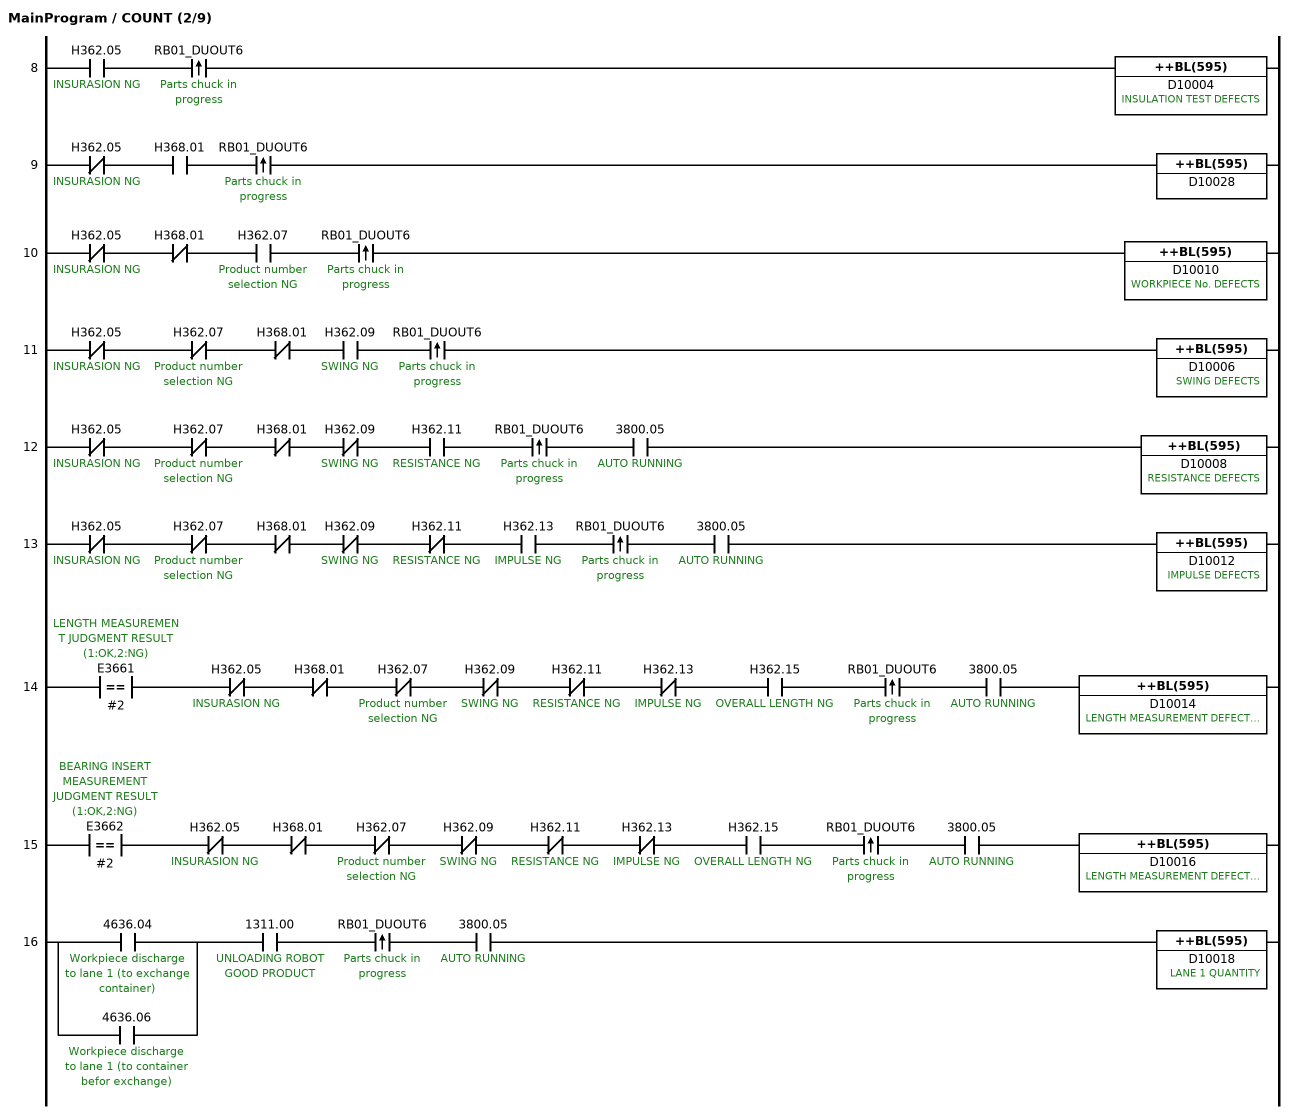
; rung 8
LD H362.05  ; INSURASION NG
@AND RB01_DUOUT6  ; Parts chuck in progress
++BL(595) D10004  ; INSULATION TEST DEFECTS
; rung 9
LDNOT H362.05  ; INSURASION NG
AND H368.01
@AND RB01_DUOUT6  ; Parts chuck in progress
++BL(595) D10028
; rung 10
LDNOT H362.05  ; INSURASION NG
ANDNOT H368.01
AND H362.07  ; Product number selection NG
@AND RB01_DUOUT6  ; Parts chuck in progress
++BL(595) D10010  ; WORKPIECE No. DEFECTS
; rung 11
LDNOT H362.05  ; INSURASION NG
ANDNOT H362.07  ; Product number selection NG
ANDNOT H368.01
AND H362.09  ; SWING NG
@AND RB01_DUOUT6  ; Parts chuck in progress
++BL(595) D10006  ; SWING DEFECTS
; rung 12
LDNOT H362.05  ; INSURASION NG
ANDNOT H362.07  ; Product number selection NG
ANDNOT H368.01
ANDNOT H362.09  ; SWING NG
AND H362.11  ; RESISTANCE NG
@AND RB01_DUOUT6  ; Parts chuck in progress
AND 3800.05  ; AUTO RUNNING
++BL(595) D10008  ; RESISTANCE DEFECTS
; rung 13
LDNOT H362.05  ; INSURASION NG
ANDNOT H362.07  ; Product number selection NG
ANDNOT H368.01
ANDNOT H362.09  ; SWING NG
ANDNOT H362.11  ; RESISTANCE NG
AND H362.13  ; IMPULSE NG
@AND RB01_DUOUT6  ; Parts chuck in progress
AND 3800.05  ; AUTO RUNNING
++BL(595) D10012  ; IMPULSE DEFECTS
; rung 14
LD=(300) E3661 #2  ; LENGTH MEASUREMENT JUDGMENT RESULT (1:OK,2:NG)
ANDNOT H362.05  ; INSURASION NG
ANDNOT H368.01
ANDNOT H362.07  ; Product number selection NG
ANDNOT H362.09  ; SWING NG
ANDNOT H362.11  ; RESISTANCE NG
ANDNOT H362.13  ; IMPULSE NG
AND H362.15  ; OVERALL LENGTH NG
@AND RB01_DUOUT6  ; Parts chuck in progress
AND 3800.05  ; AUTO RUNNING
++BL(595) D10014  ; LENGTH MEASUREMENT DEFECTS (OVERALL)
; rung 15
LD=(300) E3662 #2  ; BEARING INSERT MEASUREMENT  JUDGMENT RESULT (1:OK,2:NG)
ANDNOT H362.05  ; INSURASION NG
ANDNOT H368.01
ANDNOT H362.07  ; Product number selection NG
ANDNOT H362.09  ; SWING NG
ANDNOT H362.11  ; RESISTANCE NG
ANDNOT H362.13  ; IMPULSE NG
AND H362.15  ; OVERALL LENGTH NG
@AND RB01_DUOUT6  ; Parts chuck in progress
AND 3800.05  ; AUTO RUNNING
++BL(595) D10016  ; LENGTH MEASUREMENT DEFECTS (BEARING)
; rung 16
LD 4636.04  ; Workpiece discharge to lane 1 (to exchange container)
OR 4636.06  ; Workpiece discharge to lane 1 (to container befor exchange)
AND 1311.00  ; UNLOADING ROBOT GOOD PRODUCT
@AND RB01_DUOUT6  ; Parts chuck in progress
AND 3800.05  ; AUTO RUNNING
++BL(595) D10018  ; LANE 1 QUANTITY

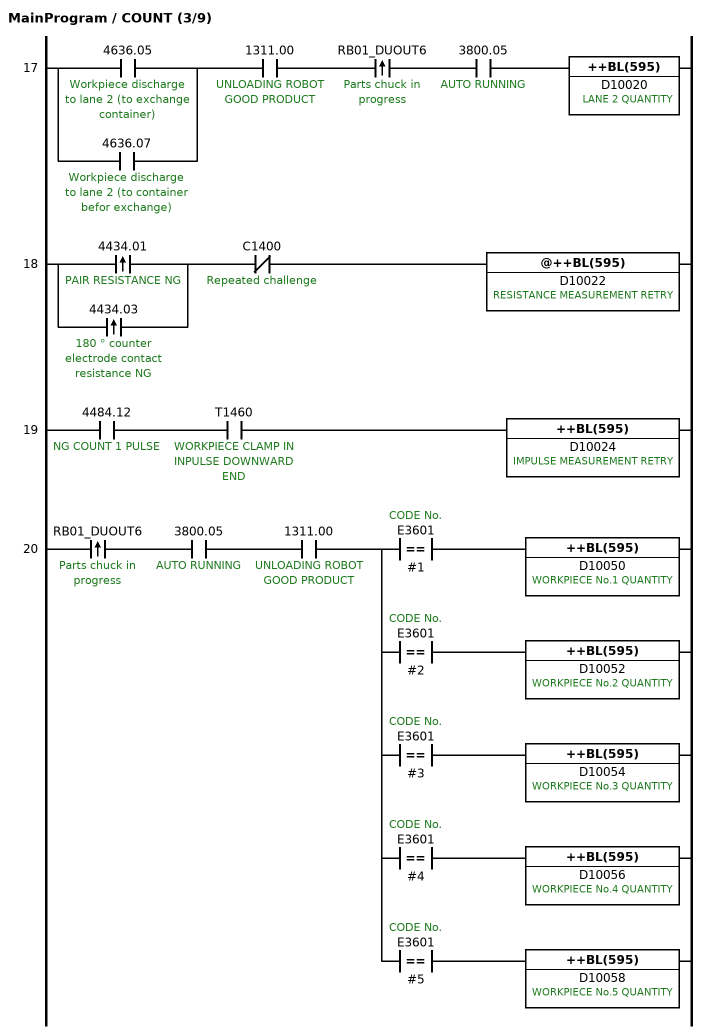
; rung 17
LD 4636.05  ; Workpiece discharge to lane 2 (to exchange container)
OR 4636.07  ; Workpiece discharge to lane 2 (to container befor exchange)
AND 1311.00  ; UNLOADING ROBOT GOOD PRODUCT
@AND RB01_DUOUT6  ; Parts chuck in progress
AND 3800.05  ; AUTO RUNNING
++BL(595) D10020  ; LANE 2 QUANTITY
; rung 18
@LD 4434.01  ; PAIR RESISTANCE NG
@OR 4434.03  ; 180 ° counter electrode contact resistance NG
ANDNOT C1400  ; Repeated challenge
@++BL(595) D10022  ; RESISTANCE MEASUREMENT RETRY
; rung 19
LD 4484.12  ; NG COUNT 1 PULSE
AND T1460  ; WORKPIECE CLAMP IN INPULSE DOWNWARD END
++BL(595) D10024  ; IMPULSE MEASUREMENT RETRY
; rung 20
@LD RB01_DUOUT6  ; Parts chuck in progress
AND 3800.05  ; AUTO RUNNING
AND 1311.00  ; UNLOADING ROBOT GOOD PRODUCT
OUT TR0
AND=(300) E3601 #1  ; CODE No.
++BL(595) D10050  ; WORKPIECE No.1 QUANTITY
LD TR0
AND=(300) E3601 #2  ; CODE No.
++BL(595) D10052  ; WORKPIECE No.2 QUANTITY
LD TR0
AND=(300) E3601 #3  ; CODE No.
++BL(595) D10054  ; WORKPIECE No.3 QUANTITY
LD TR0
AND=(300) E3601 #4  ; CODE No.
++BL(595) D10056  ; WORKPIECE No.4 QUANTITY
LD TR0
AND=(300) E3601 #5  ; CODE No.
++BL(595) D10058  ; WORKPIECE No.5 QUANTITY

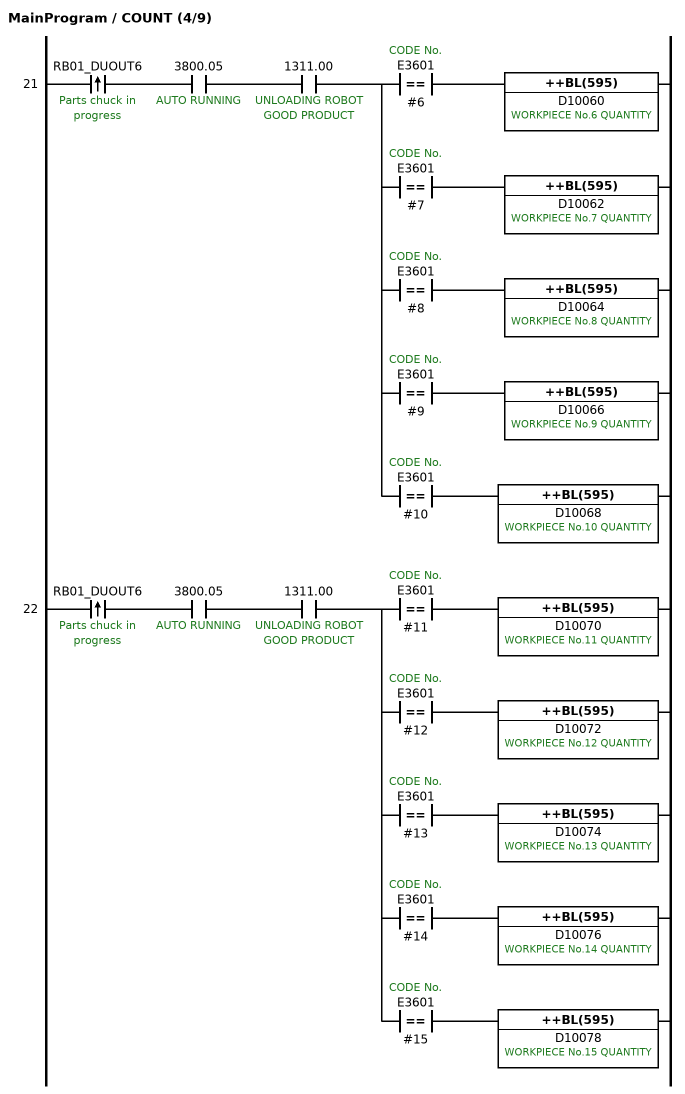
; rung 21
@LD RB01_DUOUT6  ; Parts chuck in progress
AND 3800.05  ; AUTO RUNNING
AND 1311.00  ; UNLOADING ROBOT GOOD PRODUCT
OUT TR0
AND=(300) E3601 #6  ; CODE No.
++BL(595) D10060  ; WORKPIECE No.6 QUANTITY
LD TR0
AND=(300) E3601 #7  ; CODE No.
++BL(595) D10062  ; WORKPIECE No.7 QUANTITY
LD TR0
AND=(300) E3601 #8  ; CODE No.
++BL(595) D10064  ; WORKPIECE No.8 QUANTITY
LD TR0
AND=(300) E3601 #9  ; CODE No.
++BL(595) D10066  ; WORKPIECE No.9 QUANTITY
LD TR0
AND=(300) E3601 #10  ; CODE No.
++BL(595) D10068  ; WORKPIECE No.10 QUANTITY
; rung 22
@LD RB01_DUOUT6  ; Parts chuck in progress
AND 3800.05  ; AUTO RUNNING
AND 1311.00  ; UNLOADING ROBOT GOOD PRODUCT
OUT TR0
AND=(300) E3601 #11  ; CODE No.
++BL(595) D10070  ; WORKPIECE No.11 QUANTITY
LD TR0
AND=(300) E3601 #12  ; CODE No.
++BL(595) D10072  ; WORKPIECE No.12 QUANTITY
LD TR0
AND=(300) E3601 #13  ; CODE No.
++BL(595) D10074  ; WORKPIECE No.13 QUANTITY
LD TR0
AND=(300) E3601 #14  ; CODE No.
++BL(595) D10076  ; WORKPIECE No.14 QUANTITY
LD TR0
AND=(300) E3601 #15  ; CODE No.
++BL(595) D10078  ; WORKPIECE No.15 QUANTITY

